// TwinCAT 3 PLC project iin_base
// Title: IIN_Base_T
// Company: IIN Solutions Oy
// Author: Author
// ProjectVersion: 0.0.3
// ProgramVersion: 3.1.4026.21
// libraries:
//   Tc2_Standard, * (Beckhoff Automation GmbH)
//   Tc2_System, * (Beckhoff Automation GmbH)
//   Tc2_Utilities, * (Beckhoff Automation GmbH)
//   VisuDialogs, * (System)
// project tree:
//   ALARMS/AlarmObserver/ I_AlarmObserver.TcIO
//   ALARMS/AppSupport/ FB_Interceptor.TcPOU, FB_StepperProgram.TcPOU, FC_GetLoggingId.TcPOU, FC_GetPositionWithId.TcPOU, FC_GetPosNrWithId.TcPOU, ST_INTERCEPTOR.TcDUT, ST_INTERCEPTOR_RESULT.TcDUT
//   ALARMS/DUT/ ST_ACTIVE_ALARM.TcDUT, ST_ALARM_BASE.TcDUT, ST_CLEAR_ALARM.TcDUT, ST_RAISE_ALARM.TcDUT
//   BASE/AdsUtils/ E_ADS_ERRORS.TcDUT, FC_GetAdsErrorCode.TcPOU, TL_ADS_ERRORS.TcTLO
//   BASE/ControlSignals/ FB_ControlSignalResets.TcPOU, FB_ControlSignalsV2.TcPOU, I_ControlSignals.TcIO, ST_CONTROL_SIGNALS_IN.TcDUT, ST_CONTROL_SIGNALS_OUT.TcDUT, ST_CONTROL_SIGNALS_SETTINGS.TcDUT, ST_CONTROL_SIGNALS_STATIC_SETTINGS.TcDUT, ST_CONTROL_SIGNALS_V2.TcDUT, TC_HMI_CS.TcDUT
//   BASE/CycleStartEnd/ FB_CycleEnd.TcPOU, FB_CycleStart.TcPOU, FC_GetCurrentCycleCount.TcPOU
//   BASE/FileUtils/ FC_FilePathGenerator.TcPOU
//   BASE/LocaleUtils/ E_REGIO_SELECTION.TcDUT, FB_GetLocalTimeAndDate.TcPOU, FB_TimeSync.TcPOU, FC_CallAtStart_EpochTime.TcPOU, FC_DateAndTimeToDt.TcPOU, FC_FormatTime.TcPOU, FC_GetEpochTime.TcPOU, FC_GetLocalDateAndTimeString.TcPOU, FC_GetLocalDateString.TcPOU, FC_GetLocalTimeString.TcPOU, FC_GetLocalTimeStringMinAccuracy.TcPOU, FC_GetLocalTimeStringSecAccuracy.TcPOU, FC_GetUsDateString.TcPOU, FC_NowAsDt.TcPOU, FC_TimeStringToDt.TcPOU
//   BASE/Misc/ COLORS.TcGVL, FB_Base.TcPOU, FB_BaseWithAlarmEvents.TcPOU, FB_BoolLogger.TcPOU, FB_BoolTrigger.TcPOU, FB_DelayedReset.TcPOU, FB_HandshakeDelay.TcPOU, FB_IntChangeTrigger.TcPOU, FB_IntLogger.TcPOU, FB_MemoryMonitor.TcPOU, FB_OneCycleSignalTof.TcPOU, FB_TofOnRtrig.TcPOU, FC_GetLocalAmsNetId.TcPOU, FC_GetLocalHostName.TcPOU, FC_GetMax3Arg.TcPOU, FC_GetMax3Lreals.TcPOU, FC_GetMax4Arg.TcPOU, FC_GetMin2Arg.TcPOU, FC_GetMin3Arg.TcPOU, FC_GetMin3Lreals.TcPOU, FC_GetMin4Arg.TcPOU, IING.TcGVL, ST_BASE_SETTINGS.TcDUT
//   BASE/NumberUtils/ AddREAL.TcPOU, DecINT.TcPOU, FC_CheckMinMaxInt.TcPOU, FC_CheckMinMaxReal.TcPOU, FC_KeepBetweenMinMax.TcPOU, FC_KeepBetweenMinMaxInt.TcPOU, FC_KeepRealBetweenMinMax.TcPOU, FC_LimitMaxReal.TcPOU, FC_LimitMinReal.TcPOU, FC_WithinMinMax.TcPOU, FC_WithinRange.TcPOU, IncINT.TcPOU, IncUDINT.TcPOU, IncUINT.TcPOU, IncULINT.TcPOU
//   BASE/Observer/ FB_GenericObserver.TcPOU, GVL_GENERIC_OBSERVER.TcGVL, ST_GENERIC_OBSERVER.TcDUT, ST_VALID_OBSERVERS.TcDUT
//   BASE/Persistency/ FB_Persistency.TcPOU, ST_PERSISTENCY_HMI.TcDUT, ST_PERSISTENCY_OUT.TcDUT, ST_PERSISTENCY_SERVICE.TcDUT, ST_PERSISTENCY_SETTINGS.TcDUT
//   BASE/PulsersBlinkers/ FB_Blink.TcPOU, FB_Blinkers.TcPOU, FB_Pulse.TcPOU, FB_Pulsers.TcPOU
//   BASE/StringUtils/ FC_2strConcatSeparator.TcPOU, FC_3strConcat.TcPOU, FC_3strConcatSeparator.TcPOU, FC_4strConcat.TcPOU, FC_4strConcatSeparator.TcPOU, FC_5strConcat.TcPOU, FC_5strConcatSeparator.TcPOU, FC_6strConcat.TcPOU, FC_6strConcatSeparator.TcPOU, FC_7strConcat.TcPOU, FC_7strConcatSeparator.TcPOU, FC_8strConcat.TcPOU, FC_8strConcatSeparator.TcPOU, FC_CharReplace.TcPOU, FC_FindLastOccurence.TcPOU, FC_InitializeNameAsNeeded.TcPOU, FC_IsBaseNameDefined.TcPOU, FC_LrealFormatter.TcPOU, FC_RealFormatter.TcPOU, FC_StringEmpty.TcPOU, FC_StringNotEmpty.TcPOU, FC_UintFormatter.TcPOU, IsStringEqualIgnoreCase.TcPOU
//   BASE/TypeDefinitions/ T_DEFAULT_STR.TcDUT, T_EVENT_CHAR_INDICATOR.TcDUT, T_HEART_BEAT.TcDUT, T_LONG_STR_512.TcDUT, T_SHORT_STR.TcDUT
//   DATA/DUT/ E_ALARM_REASON.TcDUT, E_ALARM_TYPE.TcDUT, E_DEVICE_TYPE.TcDUT, E_OPERATION_MODE.TcDUT, E_POS.TcDUT, E_PRIORITY.TcDUT, E_RESET_ORIGIN.TcDUT, T_DEVICE_ID.TcDUT
//   DATA/REPORTING/ DATA_REPORTER_BASE.TcGVL, FB_DummyDataReporter.TcPOU, FC_GetDataReporter.TcPOU, I_DataReporter.TcIO
//   LOGGING/ FC_GetLogger.TcPOU, LOGGER.TcGVL, NullLogger.TcPOU
//   LOGGING/FileLogger/ E_FILE_LOGGER_STEPS.TcDUT, E_FILE_SCANNER_STEPS.TcDUT, E_FILE_WRITER_STEPS.TcDUT, FB_FileLogger.TcPOU, FB_FileNameAndPath.TcPOU, FB_FileScannerV2.TcPOU, FB_FileWriterV2.TcPOU, ST_FILE_LOGGER_HMI.TcDUT, ST_FILE_LOGGER_SERVICE.TcDUT, ST_FILE_LOGGER_SETTINGS.TcDUT
//   LOGGING/GenericLogger/ FB_GenericLogger.TcPOU
//   LOGGING/NullLogger/ FB_NullLogger.TcPOU
//   LOGGING/Specs/ E_LOG_LEVEL.TcDUT, FB_LogLevel.TcPOU, I_Logger.TcIO, TL_LOG_LEVEL.TcTLO

// ---- ALARMS/AppSupport/ST_INTERCEPTOR.TcDUT
TYPE ST_INTERCEPTOR :
STRUCT
	check:	BOOL;
	desc:	T_SHORT_STR;
END_STRUCT
END_TYPE

// ---- ALARMS/AppSupport/ST_INTERCEPTOR_RESULT.TcDUT
TYPE ST_INTERCEPTOR_RESULT :
STRUCT
	clear:		BOOL;				// When TRUE, all is good 
	missing:	T_SHORT_STR;		// When clear is FALSE, this tells what is missing
END_STRUCT
END_TYPE

// ---- ALARMS/DUT/ST_ACTIVE_ALARM.TcDUT
TYPE ST_ACTIVE_ALARM EXTENDS ST_RAISE_ALARM:
STRUCT
	timestamp:				T_SHORT_STR;						// Timestamp when this occured
	epochTime:				ULINT;								// Needed for sorting purposes
	active:					BOOL;								// TRUE = currently active
END_STRUCT
END_TYPE

// ---- ALARMS/DUT/ST_ALARM_BASE.TcDUT
TYPE ST_ALARM_BASE :
STRUCT
	alarmType:			E_ALARM_TYPE := E_ALARM_TYPE.UNDEFINED;
	deviceType:			E_DEVICE_TYPE := E_DEVICE_TYPE.UNDEFINED;

	pos:				E_POS := E_POS.UNDEFINED;
	deviceId:			T_DEVICE_ID := IING.STRING_BLANK;
	
	// Unique ID generated when the alarm gets raised
	uniqueId:			ULINT;
	
	priority:			E_PRIORITY;
END_STRUCT
END_TYPE

// ---- ALARMS/DUT/ST_CLEAR_ALARM.TcDUT
TYPE ST_CLEAR_ALARM EXTENDS ST_ALARM_BASE :
STRUCT
END_STRUCT
END_TYPE

// ---- ALARMS/DUT/ST_RAISE_ALARM.TcDUT
TYPE ST_RAISE_ALARM EXTENDS ST_ALARM_BASE:
STRUCT
	givenDeviceName:		STRING;
	freeText:				STRING;
	subAlarmCode:			INT;
	
END_STRUCT
END_TYPE

// ---- BASE/AdsUtils/E_ADS_ERRORS.TcDUT
{attribute 'qualified_only'}
{attribute 'strict'}
TYPE E_ADS_ERRORS :
(
	// Global Error Codes
	NO_ERROR := 0,
	
	TARGET_PORT_NOT_FOUND := 6,
	
	TARGET_MACHINE_NOT_FOUND := 7,
	
	// General ADS Error Codes
	ADSERR_DEVICE_ERROR := 1792,
	
	ADSERR_DEVICE_SRVNOTSUPP := 1793,
	
	ADSERR_DEVICE_INVALIDGRP := 1794,
	
	ADSERR_DEVICE_INVALIDOFFSET := 1795,
	
	ADSERR_DEVICE_INVALIDACCESS := 1796,
	
	ADSERR_DEVICE_INVALIDSIZE := 1797,

	ADSERR_DEVICE_INVALIDDATA := 1798,

	ADSERR_DEVICE_NOTREADY := 1799,

	ADSERR_DEVICE_BUSY := 1800,

	ADSERR_DEVICE_INVALIDCONTEXT := 1801,

	ADSERR_DEVICE_NOMEMORY := 1802,
	
	ADSERR_DEVICE_INVALIDPARM := 1803,
	
	ADSERR_DEVICE_NOTFOUND := 1804,
	
	ADSERR_DEVICE_SYNTAX := 1805,
	
	ADSERR_DEVICE_INCOMPATIBLE := 1806,
	
	ADSERR_DEVICE_EXISTS := 1807,
	
	ADSERR_DEVICE_SYMBOLNOTFOUND := 1808,
	
	ADSERR_DEVICE_SYMBOLVERSIONINVAL := 1809,
	
	ADSERR_DEVICE_INVALIDSTATE := 1810,

	ADSERR_DEVICE_TRANSMODENOTSUPP := 1811,
	
	ADSERR_DEVICE_NOTIFYHNDINVALID := 1812,
	
	ADSERR_DEVICE_CLIENTUNKNOWN := 1813,
	
	ADSERR_DEVICE_NOMOREHDLS := 1814,
	
	ADSERR_DEVICE_INVALIDWATCHSIZE := 1815,
	
	ADSERR_DEVICE_NOTINIT := 1816,
	
	ADSERR_DEVICE_TIMEOUT := 1817,
	
	ADSERR_DEVICE_NOINTERFACE := 1818,
	
	ADSERR_DEVICE_INVALIDINTERFACE := 1819,
	
	ADSERR_DEVICE_INVALIDCLSID := 1820,
	
	ADSERR_DEVICE_INVALIDOBJID := 1821,
	
	ADSERR_DEVICE_PENDING := 1822,
	
	ADSERR_DEVICE_ABORTED := 1823,
	
	ADSERR_DEVICE_WARNING := 1824,
	
	ADSERR_DEVICE_INVALIDARRAYIDX := 1825,
	
	ADSERR_DEVICE_SYMBOLNOTACTIVE := 1826,
	
	ADSERR_DEVICE_ACCESSDENIED := 1827,
	
	ADSERR_DEVICE_LICENSENOTFOUND := 1828,
	
	ADSERR_DEVICE_LICENSEEXPIRED := 1829,
	
	ADSERR_DEVICE_LICENSEEXCEEDED := 1830,
	
	ADSERR_DEVICE_LICENSEINVALID := 1831,
	
	ADSERR_DEVICE_LICENSESYSTEMID := 1832,
	
	ADSERR_DEVICE_LICENSENOTIMELIMIT := 1833,
	
	ADSERR_DEVICE_LICENSEFUTUREISSUE := 1834,
	
	ADSERR_DEVICE_LICENSETIMETOLONG := 1835,
	
	ADSERR_DEVICE_EXCEPTION := 1836,
	
	ADSERR_DEVICE_LICENSEDUPLICATED := 1837,
	
	ADSERR_DEVICE_SIGNATUREINVALID := 1838,
	
	ADSERR_DEVICE_CERTIFICATEINVALID := 1839,
	
	ADSERR_CLIENT_ERROR := 1856,
	
	ADSERR_CLIENT_INVALIDPARM := 1857,
	
	ADSERR_CLIENT_LISTEMPTY := 1858,
	
	ADSERR_CLIENT_VARUSED := 1859,
	
	ADSERR_CLIENT_DUPLINVOKEID := 1860,
	
	ADSERR_CLIENT_SYNCTIMEOUT := 1861,
	
	ADSERR_CLIENT_W32ERROR := 1862,
	
	ADSERR_CLIENT_TIMEOUTINVALID := 1863,
	
	ADSERR_CLIENT_PORTNOTOPEN := 1864,
	
	ADSERR_CLIENT_NOAMSADDR := 1872,
	
	ADSERR_CLIENT_SYNCINTERNAL := 1873,
	
	ADSERR_CLIENT_ADDHASH := 1874,
	
	ADSERR_CLIENT_REMOVEHASH := 1875,
	
	ADSERR_CLIENT_NOMORESYM := 1876,
	
	ADSERR_CLIENT_SYNCRESINVALID := 1877,

	TODO := 9999
	
);
END_TYPE

// ---- BASE/ControlSignals/ST_CONTROL_SIGNALS_IN.TcDUT
TYPE ST_CONTROL_SIGNALS_IN :	// The raw control signals (auto/manual/service/...), do not use in your application
STRUCT
	manualMode:			BOOL;	// Auto/Manual
	serviceMode:		BOOL;
	pauseRequest:		BOOL;	// Will let ongoing operations finish nicely, When TRUE = must go to Pause, when FALSE, may continue
	stopImmediately:	BOOL;	// Placeholder for later use
	restart:			BOOL;	// Placeholder for later use
	
	reset:				BOOL;	// Reset button (a single PLC pulse will be generated from this)
	hardReset:			BOOL;	// Hard reset button (a single PLC pulse will be generated from this)

//	safetyAreaOk:		BOOL;	// Estop and doors are 'safe' = possible to drive in AUTO
	
	externalReset:		BOOL;	// External reset coming from FB_ControlSignalsV2/iExternalReset
	autoReset:			BOOL;	// Auto reset coming from FB_ControlSignalsV2/iAutoReset
END_STRUCT
END_TYPE

// ---- BASE/ControlSignals/ST_CONTROL_SIGNALS_OUT.TcDUT
TYPE ST_CONTROL_SIGNALS_OUT :	// Control signals (auto/manual/service/...) for use in programs 
STRUCT
	auto:						BOOL;	// TRUE when in automatic mode
	manual:						BOOL;	// TRUE when in manual mode
	service:					BOOL;	// TRUE when in service mode
	
	autoPulse:					BOOL;	// Single PLC cycle pulse when switching to AUTO
	manualPulse:				BOOL;	// Single PLC cycle pulse when switching to MANUAL
	servicePulse:				BOOL;	// Single PLC cycle pulse when switching to SERVICE
	
	autoOffPulse:				BOOL;	// TRUE for 1 PLC cycle when switching AUTO OFF
	manualOffPulse:				BOOL;	// TRUE for 1 PLC cycle when switching MANUAL OFF
	serviceOffPulse:			BOOL;	// TRUE for 1 PLC cycle when switching SERVICE OFF
	
	pauseRequest:				BOOL;	// TRUE when pause requested
	stopImmediately:			BOOL;	// Single PLC cycle pulse
	restart:					BOOL;	// Single PLC cycle pulse

	resetPulse:					BOOL;	// Single PLC cycle pulse for resetting (after error)
	hardResetPulse:				BOOL;	// Single PLC cycle pulse for hard reset (wipe out everything)
	
	extendedResetPulse:			BOOL;	// Extended reset pulse, eg. for external systems
	extendedHardResetPulse:		BOOL;	// Extended hard reset pulse, eg. for external systems
	
	externalManualActive:		bool;
	failingToSwitchToAuto:		BOOL;
END_STRUCT
END_TYPE

// ---- BASE/ControlSignals/ST_CONTROL_SIGNALS_SETTINGS.TcDUT
TYPE ST_CONTROL_SIGNALS_SETTINGS EXTENDS ST_BASE_SETTINGS:
STRUCT
	// All of them are under VAR_STAT
END_STRUCT
END_TYPE

// ---- BASE/ControlSignals/ST_CONTROL_SIGNALS_STATIC_SETTINGS.TcDUT
TYPE ST_CONTROL_SIGNALS_STATIC_SETTINGS:
STRUCT
	resetTime:						TIME := IING.RESET_TIME;
	hardResetTime:					TIME := IING.HARD_RESET_TIME;
	serviceResetTime:				TIME := IING.AUTO_SERVICE_RESET_TIME;	// Time after which service mode is swithced OFF
	extendedResetPulseDuration:		TIME := IING.EXTENDED_RESET_PULSE_DURATION;
END_STRUCT
END_TYPE

// ---- BASE/ControlSignals/ST_CONTROL_SIGNALS_V2.TcDUT
TYPE ST_CONTROL_SIGNALS_V2 :	// Control signals (auto/manual/service/...) for use in programs 
STRUCT
	in:				 	ST_CONTROL_SIGNALS_IN;
	out:				ST_CONTROL_SIGNALS_OUT;
	
	settings:			REFERENCE TO ST_CONTROL_SIGNALS_SETTINGS;
	staticSettings:		REFERENCE TO ST_CONTROL_SIGNALS_STATIC_SETTINGS;
END_STRUCT
END_TYPE

// ---- BASE/ControlSignals/TC_HMI_CS.TcDUT
TYPE TC_HMI_CS :
STRUCT
	out:		ST_CONTROL_SIGNALS_OUT;
	in:	ST_CONTROL_SIGNALS_IN;
END_STRUCT
END_TYPE

// ---- BASE/LocaleUtils/E_REGIO_SELECTION.TcDUT
{attribute 'qualified_only'}
{attribute 'strict'}
TYPE E_REGIO_SELECTION :
(
	USA := 0,
	EUROPE
);
END_TYPE

// ---- BASE/Misc/ST_BASE_SETTINGS.TcDUT
TYPE ST_BASE_SETTINGS :
STRUCT
	name:			T_SHORT_STR := IING.STRING_BASE_SETTINGS_INITIAL_NAME;
	doHide:			BOOL := TRUE;
END_STRUCT
END_TYPE

// ---- BASE/Observer/ST_GENERIC_OBSERVER.TcDUT
TYPE ST_GENERIC_OBSERVER :
STRUCT
	who:		T_SHORT_STR;			// Unique identifier of this observer
	observer:	POINTER TO BYTE;		// Interface CASTed to a generic POINTER, to be CASTed back in your application
END_STRUCT
END_TYPE

// ---- BASE/Observer/ST_VALID_OBSERVERS.TcDUT
TYPE ST_VALID_OBSERVERS :
STRUCT
	cnt:		INT;
	observers:	ARRAY[0..GVL_GENERIC_OBSERVER.OBSERVER_CNT-1] OF ST_GENERIC_OBSERVER;
END_STRUCT
END_TYPE

// ---- BASE/Persistency/ST_PERSISTENCY_HMI.TcDUT
TYPE ST_PERSISTENCY_HMI :
STRUCT
	service:		REFERENCE TO ST_PERSISTENCY_SERVICE;
	settings:		REFERENCE TO ST_PERSISTENCY_SETTINGS;
	out:			REFERENCE TO ST_PERSISTENCY_OUT;
END_STRUCT
END_TYPE

// ---- BASE/Persistency/ST_PERSISTENCY_OUT.TcDUT
TYPE ST_PERSISTENCY_OUT :
STRUCT
	busy:					BOOL;
	error:					BOOL;
	beckhoffErrorId:		UDINT;
	errorIdEnum:			E_ADS_ERRORS;
END_STRUCT
END_TYPE

// ---- BASE/Persistency/ST_PERSISTENCY_SERVICE.TcDUT
TYPE ST_PERSISTENCY_SERVICE :
STRUCT
	saveNow:		BOOL;
END_STRUCT
END_TYPE

// ---- BASE/Persistency/ST_PERSISTENCY_SETTINGS.TcDUT
TYPE ST_PERSISTENCY_SETTINGS :
STRUCT
	port:				UINT := 851;	
	autoSave:			BOOL := TRUE;
	saveInterval:		TIME := T#12H;
END_STRUCT
END_TYPE

// ---- BASE/TypeDefinitions/T_DEFAULT_STR.TcDUT
TYPE T_DEFAULT_STR : STRING(255); END_TYPE		// Use this instead of STRING which is 80 chars only

// ---- BASE/TypeDefinitions/T_EVENT_CHAR_INDICATOR.TcDUT
TYPE T_EVENT_CHAR_INDICATOR : STRING(1); END_TYPE

// ---- BASE/TypeDefinitions/T_HEART_BEAT.TcDUT
TYPE T_HEART_BEAT : UDINT; END_TYPE		// Signal used to check the heart beat (over ADS)

// ---- BASE/TypeDefinitions/T_LONG_STR_512.TcDUT
TYPE T_LONG_STR_512 : STRING(512); END_TYPE		// Use this instead of STRING which is 80 chars only

// ---- BASE/TypeDefinitions/T_SHORT_STR.TcDUT
TYPE T_SHORT_STR : STRING(80); END_TYPE		// Use this for 'shorter' string

// ---- DATA/DUT/E_ALARM_REASON.TcDUT
{attribute 'qualified_only'}

{attribute 'to_string'}
TYPE E_ALARM_REASON :
(
	UNDEFINED,
	
	NO_COOLING,
	
	OVERLOAD,
	
	WRONG_ITEM,
	
	WRONG_DIMENSION,
	
	WRONG_ORIENTATION,
	
	STUCK,
	
	NO_PRESSURE,
	
	OTHER,	
	
	MUST_BE_LAST	// ALWAYS KEEP THIS LAST!!!
	
);
END_TYPE

// ---- DATA/DUT/E_ALARM_TYPE.TcDUT
{attribute 'qualified_only'}
{attribute 'to_string'}
TYPE E_ALARM_TYPE :
(
	UNDEFINED := 0,

	// An operation took too long to complete
	TIME_OUT,

	// A sensor is blocked
	SENSOR_BLOCKED,
	
	// Bad request, eg. asking to open and close a cylinder at the same time 
	BAD_REQUEST,
	
	// Overload from eg. a fuse or servo drive
	OVERLOAD,
	
	// A component is overheating
	OVERHEAT,

	// Collision detected
	COLLISION,
	
	// Regular servo error
	SERVO_ERROR,
	
	// Positioning error
	POSITIONING_ERROR,
	
	// Velocity error
	VELOCITY_ERROR,
	
	MOVE_RELATIVE_ERROR,
	
	// Jogging error
	JOGGING_ERROR,

	// Probing error	
	PROBING_ERROR,
	
	// Gearing error
	GEARING_ERROR,
	
	GEAR_IN_ERROR,
	
	GEAR_OUT_ERROR,
	
	// Measurement of a member/truss did not match the WP length
	DIMENSION_MISMATCH,
	
	// Buffer station or robots get values not in the allowed work area
	WRONG_COORDINATES,
	
	// Member id (or eventId) mismatch, plate mismatch
	ITEM_MISMATCH,
	
	ESTOP,
	
	BELOW_MIN,
	
	ABOVE_MAX,
	
	// Communication error
	COMM_ERROR,
	
	MISSING_PART,
	
	HOMING_ERROR,
	
	ZEROING_ERROR,
	
	TOOL_DROP,
	
	SAFETY,
	
	DOCKING_STATION_ERROR,
	
	PARSE_ERROR,
	
	TOOL_CHANGER_ERROR,
	
	// Sequence expects something but this is not fullfilled
	WRONG_STATE,
	
	HOMING_NOT_ENABLED,
	
	// Eg, not supported settings (nor head, nor tail selection)
	CONFIGURATION_ERROR,

	FORCING,			// Used with the Forcing alarm manager
	
	NO_POWER,			// Power supply 'OFF'
	
	INTERRUPTION,		// Something got interrupted/stopped, eg. STOPMESS in robot

	TASK_DIED,			// Eg. submit interpreter not running
	
	SIMULATION_ACTIVE,
	
	STICKY_BUTTON,		// Eg. a button is sticky (PLC HMI)
	
	SAFE_TORQUE_OFF,	// STO active, eg, freq drive or servo
	
	FREQ_DRIVE_ERROR,	// Any kind of frequence related error

	START_CONDITIONS_NOT_MET,
	
	MISC,
	
	OUT_OF_RANGE,
	
	CLOGGED,					// Eg. filter clogged
	
	MISSING,					// Eg. air pressure missing
	
	OPEN,						// Eg. a door is open
	
	PREMATURE_DETECTION,		// Probing ready before slowing down conveyor
	
	TRIGGERED,					// Safety scanner got triggered
	
	LOW_VALUE,					// eg. speed setting rather low, intentional?
	
	DEVIATION_DETECTED,			// AI and AO settings not matching (enfield)
	
	OVERSHOOTING,				// Servo is overshooting (then reversing)
	
	SENSOR_BROKEN,				// AI readings not possible
	
	ROBOT_APP_ERROR,			// Robot sends us some error code (probably calculation/e1 related)
	
	VACUUM_MISSING,				// Vacuum is missing
	
	MANUAL_MODE,				// Device is in manual
	
	EDM,						// External Device Monitoring
	
	CLOSED,						// Eg. a (gantry) door is closed
	
	WAITING_CONFIRMATION,
	
	SUPER_POWERS,
	
	END //63
	
);
END_TYPE

// ---- DATA/DUT/E_DEVICE_TYPE.TcDUT
{attribute 'qualified_only'}

{attribute 'to_string'}
TYPE E_DEVICE_TYPE :
(
	UNDEFINED,
	
	// Special case for alarm handler	
	ACCEPT_ANY,
	
	MOTOR,					// Direct drive motor

	SERVO,					// Servo drive
	
	FREQ_DRIVE,				// 'TAMU'

	FUSE,
	
	RELAIS,
	
	VALVE,
	
	CYLINDER,
	
	HYDRAULIC,
	
	SCANNER,				// Eg. sick scanner		

	PRINTER,		
	
	DOOR,					// Eg. Safety door
	
	ESTOP,
	
	BRAKE,
	
	PSU,
	
	FILTER,					// Eg. oil/air filter
	
	CONVEYOR,
	
	COMM_CHANNEL,
	
	TURN_TABLE,
	
	MISC,
	
	ROBOT,
	
	MAGNET,
	
	SENSOR,		// Use this for
	
	SPEED_CONTROL,	// Device speed
	
	TOOL_CHANGER,
	
	BUTTON_BOX,
	
	PNEUMATIC,
	
	SAFETY,
	
	ENCODER,
	
	SEQUENCE,
	
	CONTROL_SIGNALS,
	
	END	// ALWAYS KEEP THIS LAST!!!
);
END_TYPE

// ---- DATA/DUT/E_OPERATION_MODE.TcDUT
{attribute 'qualified_only'}
{attribute 'strict'}
{attribute 'to_string'}
TYPE E_OPERATION_MODE :
(
	UNDEFINED,
	
	AUTO,

	MANUAL,
	
	MUST_BE_LAST	// ALWAYS KEEP THIS LAST!!!
);
END_TYPE

// ---- DATA/DUT/E_POS.TcDUT
{attribute 'qualified_only'}
{attribute 'to_string'}
TYPE E_POS :			// Position numbers
(
	UNDEFINED := 0,
	
	// Special case for alarm handler	
	ACCEPT_ANY := 1,

	MAIN :=		10,
	

	
	
	MUST_BE_LAST	// ALWAYS KEEP THIS LAST!!!
);
END_TYPE

// ---- DATA/DUT/E_PRIORITY.TcDUT
{attribute 'qualified_only'}
{attribute 'strict'}
{attribute 'to_string'}
TYPE E_PRIORITY :
(
	UNDEFINED,
	
	LOW,
	
	MEDIUM,
	
	HIGH,
	
	MUST_BE_LAST	// ALWAYS KEEP THIS LAST!!!
);
END_TYPE

// ---- DATA/DUT/E_RESET_ORIGIN.TcDUT
{attribute 'qualified_only'}
{attribute 'strict'}
{attribute 'to_string'}
TYPE E_RESET_ORIGIN :
(
	UNDEFINED := 0,
	
	CONTROL_AREA_MANUAL,	// Operator presses reset on the control signal
	
	CONTROL_AREA_AUTO,		// Automatic (external) reset, eg. doors were closed and a reset was triggered

	EXTERNAL,				// Through FB input, eg. hard wired button or banner reset
	
	ALARM_SPECIFIC			// Specific device/alarm reset 
);
END_TYPE

// ---- DATA/DUT/T_DEVICE_ID.TcDUT
TYPE T_DEVICE_ID : STRING; END_TYPE

// ---- LOGGING/FileLogger/E_FILE_LOGGER_STEPS.TcDUT
{attribute 'qualified_only'}
{attribute 'strict'}
TYPE E_FILE_LOGGER_STEPS :
(
	WAIT_ACTIVITY := 0,
	
	CHECK_SIZE,
	
	CLOSE_FILE,
	
	SCAN_FOLDER,
	
	ITERATE_FILES,
	
	RENAME_FILE,
	
	RENAME_FILE_ERROR,
	
	END
);
END_TYPE

// ---- LOGGING/FileLogger/E_FILE_SCANNER_STEPS.TcDUT
{attribute 'qualified_only'}
{attribute 'strict'}
TYPE E_FILE_SCANNER_STEPS :
(
	IDLE := 0,
	
	SCAN,
	
	STORE_FILE,
	
	DONE,
	
	ERROR,
	
	END
);
END_TYPE

// ---- LOGGING/FileLogger/E_FILE_WRITER_STEPS.TcDUT
{attribute 'qualified_only'}
{attribute 'strict'}
TYPE E_FILE_WRITER_STEPS :
(
	IDLE := 0,
	
	OPEN_FILE,
	
	WAIT_DATA,
	
	WRITE_LINE,

	CHECK_FILE,
	
	CLOSE_FILE,
	
	CLEANUP,
	
	OPENING_ERROR,
	
	TELL_ERROR,
	
	WRITING_ERROR,
	
	CLOSING_ERROR,
	
	END
);
END_TYPE

// ---- LOGGING/FileLogger/ST_FILE_LOGGER_HMI.TcDUT
TYPE ST_FILE_LOGGER_HMI :
STRUCT
	// Modifiable from HMI
	service:					REFERENCE TO ST_FILE_LOGGER_SERVICE;
	settings:					REFERENCE TO ST_FILE_LOGGER_SETTINGS;	
	controlSignals:				REFERENCE TO ST_CONTROL_SIGNALS_IN;

	amsNetId:					T_AmsNetId;
	fileNameAndPath:			T_DEFAULT_STR;					// VISU helper
	tracingOn:					BOOL;							// TRUE when log level is trace
	tracingTimeExpired:			TIME;							// Amount of trace time expired
	autoResetOn:				BOOL;							// TRUE when auto reset is ON
	outResetTimer:				TIME;							// After this time, auto reset will be done
	error:						BOOL;							// TRUE if a file writing error occurs
	adsErrorCode:				E_ADS_ERRORS;
	fileWriterRecordCnt:		UDINT;
	fileWriterBytesUsed:		UDINT;
	fileWriterOverflowCount:	UDINT;							// How many times we were not able to write all data to the file (due to internal memory constraints)
END_STRUCT
END_TYPE

// ---- LOGGING/FileLogger/ST_FILE_LOGGER_SERVICE.TcDUT
TYPE ST_FILE_LOGGER_SERVICE :
STRUCT
	doFileFlush:			BOOL;							// Set TRUE when flush is wanted
END_STRUCT
END_TYPE

// ---- LOGGING/FileLogger/ST_FILE_LOGGER_SETTINGS.TcDUT
TYPE ST_FILE_LOGGER_SETTINGS EXTENDS ST_BASE_SETTINGS:
STRUCT
	logLevel:				E_LOG_LEVEL := E_LOG_LEVEL.ERROR;	// The current log level
	maxFileSizeMB:			DINT := 10;							// File size (MB) after which, the log file will be rolled over
	enableMaxTracingTime:	BOOL := FALSE;						// When TRUE, TRACING can be switched off automatically
	maxTracingTime:			TIME := T#1H;						// Max amount of time TRACING will be active, after this DEBUG becomes activeEND_STRUCT
	enableAutoReset:		BOOL := TRUE;						// When TRUE, write errors will be reset automatically
	autoResetTime:			TIME := T#1H;						// After this amount of time, an error reset will be done
END_STRUCT
END_TYPE

// ---- LOGGING/Specs/E_LOG_LEVEL.TcDUT
{attribute 'qualified_only'}
{attribute 'strict'}
{attribute 'to_string'}
TYPE E_LOG_LEVEL :
(
	TRACE := 0,			// Use for hard to find problems = tracing problems, this will generate a log of data
	
	DEBUG,			// Debug logging (steps)
	
	INFO,			// Use for informational messages
	
	WARN,			// Use for warnings
	
	ERROR,			// Use for errors/alarms

	OFF			// Nothing will be logged
);
END_TYPE

// ---- BASE/Misc/COLORS.TcGVL
{attribute 'qualified_only'}
{attribute 'global_init_slot' := '40001'}
VAR_GLOBAL CONSTANT
	LILA:	DWORD := 16#FF0F0DF1;
	PINK:	DWORD := 16#FFE943D4;
	ORANGE:	DWORD := 16#FFFFCC00;
	BLUE :	DWORD := 16#FF0000FF;
	RED	:	DWORD := 16#FFFF0000;
	YELLOW:	DWORD := 16#FFFFFF00;
	GREEN:	DWORD := 16#FF00FF00;
	GREY:	DWORD := 16#FFC0C0C0;
	WHITE:	DWORD := 16#FFFFFFFF;
	BLACK:	DWORD := 16#FF000000;	
END_VAR

// ---- BASE/Misc/IING.TcGVL
{attribute 'qualified_only'}
{attribute 'global_init_slot' := '40002'}
VAR_GLOBAL
	epochtime :						ULINT;				// Epoch time (milliseconds)
	localSystemTime:				TIMESTRUCT;			// Local system time
	localDateString:				T_SHORT_STR;		// Local date string, eg. '27:5:2019'. Use E_REGIO_SELECTION at FB_CycleStart for a different format.
	usDateString:					T_SHORT_STR;		// US style date string, especially usefull for naming log files
	localTimeString:				T_SHORT_STR;		// Local time as string, eg. '15:58:40:302'
	localDateAndTimeString:			T_SHORT_STR;		// Local date and time as string,  eg. '27:5:2019 15:58:40:302'. Use E_REGIO_SELECTION at FB_CycleStart for a different format.
	localHostName:					T_DEFAULT_STR;		// Local hostname
	localAmsNetId:					T_AmsNetId;			// Local AMS net id
	localTimeSecAccuracy:			T_SHORT_STR;		// Local time as string, eg. '15:58:40', seconds accuracy
	localTimeMinAccuracy:			T_SHORT_STR;		// Local time as string, eg. '15:58', minutes accuracy
	iso8601Time:					T_SHORT_STR;		// Time in ISO 8601 format
	
	cycleTime:						ULINT;				// Current PLC cycle time in msec
	cycleStart:						BOOL;				// TRUE during first PLC cycle
	lastPlcRestart:					T_SHORT_STR;		// Timestamp of last PLC restart
	dayHasChanged:					BOOL;				// TRUE for 1 PLC cycle when a day change occurs

	// Blinkers, usefull for making a light beacon blink
	blink100Ms:						BOOL;			// 100ms blinker  
	blink500Ms:						BOOL;			// 500ms blinker
	blink1S:						BOOL;			// 1S blinker
	blink2S:						BOOL;			// 2S blinker
	blink5S:						BOOL;			// 5S blinker
	blink10S:						BOOL;			// 10S blinker
	
	invertedBlink100Ms:				BOOL;			// Inverted 100ms blinker
	invertedBlink500Ms:				BOOL;			// Inverted 500ms blinker
	invertedBlink1S:				BOOL;			// Inverted 1S blinker
	invertedBlink2S:				BOOL;			// Inverted 2S blinker
	invertedBlink5S:				BOOL;			// Inverted 5S blinker
	invertedBlink10S:				BOOL;			// Inverted 10S blinker
 
	// 1 'PLC cycle' long pulsers 
	pulse100Ms:						BOOL;
	pulse500Ms:						BOOL;
	pulse1S:						BOOL;
	pulse2S:						BOOL;
	pulse10S:						BOOL;
	pulse30S:						BOOL;
	pulse1M:						BOOL;
	pulse1H:						BOOL;
	
	STRING_EMPTY_NON_CONSTANT:		T_SHORT_STR := '';			// Some VISUs want write access
	cycleCounter:					UDINT;			// Gets incremented each PLC cycle
	adsPort:						UINT;			// The ADS port we are running on
	
	simulatorActive:				BOOL;		// TRUE when running in simulation mode (TC project variant 'simulator')
	pointerSize:					UINT;		// Number of bytes for a pointer (=size)
END_VAR

VAR_GLOBAL CONSTANT
	TIME_OFFSET_1601 : 				ULINT := 11644472389000;	// Jan 01, 1601 (gotten from online millisecond calculator)
	TIME_OFFSET_20MINS :			ULINT := 20 *60 *1000;		// 1601 offset is 20 mins WRONG!
	EPOCH_CORRECTION :				ULINT := TIME_OFFSET_1601 + TIME_OFFSET_20MINS;		// Correction to get proper EPOCH timestamp instead of Beckhoff timestamp
	
	STRING_BLANK:					T_SHORT_STR := '';				// Use this instead of '', renamed from EMPTY->BLANK since same string exist in Beckhoff libs
	STRING_COLON: 					T_SHORT_STR := ':';				// Use this instead of ':'
	STRING_SPACE: 					T_SHORT_STR := ' ';				// Use this instead of ' '
	STRING_UNDERSCORE:				T_SHORT_STR := '_';				// Use this instead of '_'
	STRING_DASH:					T_SHORT_STR := '-';				// Use this instead of '-'
	STRING_COMMA:					T_SHORT_STR := ',';				// Use this instead of ','
	STRING_STAR:					T_SHORT_STR := '*';				// Use this instead of '*'
	STRING_SLASH:					T_SHORT_STR := '/';				// Use this instead of '/'
	STRING_BACKSLASH:				T_SHORT_STR := '\';				// Use this instead of '\'
	STRING_SQUARE_BRACKET_OPEN:		T_SHORT_STR := '[';				// Use this instead of '['
	STRING_SQUARE_BRACKET_CLOSE:	T_SHORT_STR := ']';				// Use this instead of ']'
	STRING_DOT:						T_SHORT_STR := '.';				// Use this instead of '.'
	STRING_PIPE:					T_SHORT_STR := '|';				// Use this instead of '|'
	STRING_AM:						T_SHORT_STR := 'AM';			// Use for time formatting
	STRING_PM:						T_SHORT_STR := 'PM';			// Use for time formatting
	STRING_BASE_SETTINGS_INITIAL_NAME:	T_SHORT_STR := '???';	// Initial name for the base setting
	STRING_EQUALS:					T_SHORT_STR := '=';				// Use this instead of '='
	STRING_EXCLAMATION:				T_SHORT_STR := '!';				// Use this instead of '!'
	STRING_UNDEFINED:				STRING := 'undefined';
	
	
	
	STRING_LINE_FEED:				T_SHORT_STR := '$0A';			// Use this when adding a line feed (eg. file handling)
	
	STRING_80_CHARS:				T_SHORT_STR := '0123456789012345678901234567890123456789012345678901234567890123456789012345678_';	// Use this for testing string functions (string by default is 80 chars only)
	STRING_TODO:					T_SHORT_STR := 'TODO';
	
	ADS_WRITE_TIMEOUT:				TIME := T#1S;				// Default ADS time-out for our applications
	ADS_WRITE_RETRIES:				UDINT := 3;					// Default number of ADS retries
	ADS_DEFAULT_PORT:				T_AmsPort := 851;			// Default ADS port (for 1st PLC)
	ADS_MB_INDEX_GROUP:				UDINT := 16#4020;			// ADS MB index group
	
	IDX_UNDEFINED:					INT := -1;					// Use this to make an array index invalid (instead of just 0)
	INVALID_UINT:					INT := -1;					// Use this to make an UINT invalid (instead of just 0)
	
	RESET_TIME:						TIME := T#100MS;			// Normal reset default time/delay
	HARD_RESET_TIME:				TIME := T#1S;				// Hard reset default time/delay
	AUTO_SERVICE_RESET_TIME:		TIME := T#5M;				// Time after which service mode is switched OFF
	EXTENDED_RESET_PULSE_DURATION:	TIME := T#250MS;
	SERVO_POWER_SAVINGS_TIME:		TIME := T#5M;				// Automatic powering down of a SERVO	
	
	BITS_IN_WORD:					UINT := 16;					// Number of bits in a WORD
	BITS_IN_DWORD:					UINT := 32;					// Number of bits in a DWORD
	
	FULL_SPEED:						REAL := 100.0;				// Use this as the default velocity override speed
	
	ZERO_POINTER:					UDINT := 0;					// Use this to 'null' a pointer/reference
	ONE_INCH:						LREAL := 25.4;				// One inch

	ONE_KBYTE:						DINT := 1024;				// One kilobyte in bytes	
	ONE_MBYTE:						DINT := 1048576;			// One megabyte in bytes
	
	MAX_UDINT:						UDINT := 16#FFFFFFFF;		// Biggest possible UDINT
	MAX_INT:						INT := 32767;				// Max value for an INT

	EVENT_INDICATION_NONE:			T_EVENT_CHAR_INDICATOR := STRING_BLANK;
	EVENT_INDICATION_WARNING:		T_EVENT_CHAR_INDICATOR := 'W';
	EVENT_INDICATION_ALARM:			T_EVENT_CHAR_INDICATOR := 'A';	
END_VAR

// ---- BASE/Observer/GVL_GENERIC_OBSERVER.TcGVL
{attribute 'qualified_only'}
VAR_GLOBAL CONSTANT
	OBSERVER_CNT:	INT := 5;
END_VAR

// ---- DATA/REPORTING/DATA_REPORTER_BASE.TcGVL
{attribute 'qualified_only'}
VAR_GLOBAL
	dummyReporter:		FB_DummyDataReporter;
	defaultReporter:	I_DataReporter;
END_VAR

// ---- LOGGING/LOGGER.TcGVL
{attribute 'qualified_only'}
VAR_GLOBAL
	nullLogger:				FB_NullLogger;					// DEV 0 logger
	defaultLogger:			I_Logger;	
END_VAR

// ---- ALARMS/AlarmObserver/I_AlarmObserver.TcIO
INTERFACE I_AlarmObserver

METHOD PUBLIC cleared : BOOL		// Called when an alarm is cleared
VAR_INPUT
	iAlarm:	ST_CLEAR_ALARM;
END_VAR
END_METHOD

METHOD PUBLIC raised : BOOL		// Called when an alarm is raised
VAR_INPUT
	iAlarm:	ST_ACTIVE_ALARM;
END_VAR
END_METHOD

END_INTERFACE

// ---- BASE/ControlSignals/I_ControlSignals.TcIO
INTERFACE I_ControlSignals

METHOD ic_getControlSignalsOutPtr : POINTER TO ST_CONTROL_SIGNALS_OUT
END_METHOD

METHOD PUBLIC ic_getControlSignalsPtr : POINTER TO ST_CONTROL_SIGNALS_V2
END_METHOD

METHOD PUBLIC ic_isInAuto : BOOL
END_METHOD

METHOD PUBLIC ic_isInPause : BOOL
END_METHOD

METHOD PUBLIC ic_switchToAuto
END_METHOD

METHOD ic_unPause
END_METHOD

END_INTERFACE

// ---- DATA/REPORTING/I_DataReporter.TcIO
INTERFACE I_DataReporter		// Interface for all data/mqtt reporting calls.
	// Idea is to keep logic away from the project/application, also reporting can be done in several ways, such as mqtt

METHOD PUBLIC ic_deviceSpeedChanged	// To be called when the (device) speed changes
VAR_INPUT
	iPos:			E_POS;				// Position enumerate
	iMiscArea:		T_SHORT_STR;		// Safety or misc area enumerate (string). If defined/non-empty, use this instead of iPos
	iNew:			INT;				// The new speed value
END_VAR
END_METHOD

METHOD PUBLIC ic_initializeDone	// To be called when a initialization (aka hard reset) is done
VAR_INPUT
	iPos:			E_POS;				// The position
	iMiscArea:		T_SHORT_STR;		// Safety or misc area enumerate (string). If defined/non-empty, use this instead of iPos
	iOrigin:		E_RESET_ORIGIN;	
END_VAR
END_METHOD

METHOD PUBLIC ic_operationModeChanged	// To be called when the control signal operation mode changes
VAR_INPUT
	iPos:			E_POS;				// The position
	iMiscArea:		T_SHORT_STR;		// Safety or misc area enumerate (string). If defined/non-empty, use this instead of iPos
	iNew:			E_OPERATION_MODE;	// New operation mode
END_VAR
END_METHOD

METHOD PUBLIC ic_resetDone	// To be called when the control signal operation mode changes
VAR_INPUT
	iPos:			E_POS;				// The position
	iMiscArea:		T_SHORT_STR;		// Safety or misc area enumerate (string). If defined/non-empty, use this instead of iPos
	iOrigin:		E_RESET_ORIGIN;
	iResetKeyLabel:	T_SHORT_STR;		// What reset key was pressed
END_VAR
END_METHOD

METHOD PUBLIC ic_serviceStateChanged		// To be called when the (control signal) service state changes
VAR_INPUT
	iPos:			E_POS;				// The position
	iMiscArea:		T_SHORT_STR;		// Safety or misc area enumerate (string). If defined/non-empty, use this instead of iPos
	iState:			BOOL;				// TRUE = service activated, FALSE = service deactivated
END_VAR
END_METHOD

END_INTERFACE

// ---- LOGGING/Specs/I_Logger.TcIO
INTERFACE I_Logger		// Generic interface for logging 'data', logging can be done to file/HMI/MQTT and depends on the implementation

METHOD PUBLIC debug : BOOL	// Logs the data with log level 'DEBUG'
VAR_INPUT
	iData:		T_DEFAULT_STR;						// Data to be logged, limited to 255 characters
END_VAR
END_METHOD

METHOD PUBLIC deregister : BOOL
VAR_INPUT
	iWho:				T_SHORT_STR;
END_VAR
END_METHOD

METHOD PUBLIC doLog : BOOL	// Logs the data with log level iLevel
VAR_INPUT
	iData:		T_DEFAULT_STR;						// Data to be logged, limited to 255 characters
	iLevel:		E_LOG_LEVEL := E_LOG_LEVEL.ERROR;	// Log level
END_VAR
END_METHOD

METHOD PUBLIC error : BOOL	// Logs the data with log level 'ERROR'
VAR_INPUT
	iData:		T_DEFAULT_STR;						// Data to be logged, limited to 255 characters
END_VAR
END_METHOD

METHOD PUBLIC info : BOOL	// Logs the data with log level 'INFO'
VAR_INPUT
	iData:		T_DEFAULT_STR;						// Data to be logged, limited to 255 characters
END_VAR
END_METHOD

METHOD PUBLIC register : BOOL
VAR_INPUT
	iWho:		T_SHORT_STR;
	iObserver:	I_Logger;
END_VAR
END_METHOD

METHOD PUBLIC trace : BOOL	// Logs the data with log level 'TRACE'
VAR_INPUT
	iData:		T_DEFAULT_STR;						// Data to be logged, limited to 255 characters
END_VAR
END_METHOD

METHOD PUBLIC warn : BOOL	// Logs the data with log level 'WARN'
VAR_INPUT
	iData:		T_DEFAULT_STR;						// Data to be logged, limited to 255 characters
END_VAR
END_METHOD

END_INTERFACE

// ---- BASE/CycleStartEnd/FB_CycleStart.TcPOU
FUNCTION_BLOCK FB_CycleStart		// Must always be the 1st call in PLC MAIN, ensures other functions/globals are available 
VAR_INPUT
	iRegioSelection:		E_REGIO_SELECTION := E_REGIO_SELECTION.USA;		// Regio selection, will affect to date/time formatting
	iLogger:				I_Logger := NullLogger();
END_VAR
VAR_OUTPUT
	
	oPersistencyHmi:		ST_PERSISTENCY_HMI;
END_VAR
VAR
	getHostName: 			FB_GetHostName;
	getAmsNetId:			FB_GetLocalAmsNetId;
	
	getLocalTime: 			FB_GetLocalTimeAndDate;
	
	blinkers:				FB_Blinkers;
	pulsers:				FB_Pulsers;
	
	
	persistency:			FB_Persistency;
	
	taskIndex:				DINT;		// The task index of the task in which we are called.
	
	pointerToByte:			POINTER TO BYTE;
END_VAR
VAR PERSISTENT
	numberOfPlcStarts:		UDINT;	// How often the PLC has been started
	timeOfPreviousCycle:	ULINT;
END_VAR

// Read epoch time
FC_CallAtStart_EpochTime();

// Read local system time as string
getLocalTime(iRegioSelection := iRegioSelection);

// Was used earlier to determine the cycleStart flag
IING.cycleTime := FC_GetEpochTime() - timeOfPreviousCycle;

// The famous cycle start flag, earlier done by checking the cycle time, TTECH-4497
taskIndex := GETCURTASKINDEXEX();	// -1 = The function is called from the Windows context.
									// 0 = The function is called from the real-time context, but not from a cyclic PLC task. This is the case, for example, with the automatic call of FB_init methods during initialization.
									// 1 to n = The function is called from a cyclic PLC task. The return value is the task index.
IF (taskIndex > 0) THEN
	IING.cycleStart :=  TwinCAT_SystemInfoVarList._TaskInfo[taskIndex].FirstCycle;
	IING.cycleCounter := TwinCAT_SystemInfoVarList._TaskInfo[taskIndex].CycleCount;
	IING.adsPort := TwinCAT_SystemInfoVarList._TaskInfo[taskIndex].AdsPort;
ELSE
	IING.cycleStart := FALSE;
	IING.cycleCounter := 0;
END_IF

IF (IING.cycleStart) THEN
	IncUDINT(numberOfPlcStarts);
	
	IING.pointerSize := SIZEOF(pointerToByte);
END_IF
timeOfPreviousCycle := FC_GetEpochTime();

// Read host name and AMS net id
getHostName(bExecute := IING.cycleStart, tTimeout := DEFAULT_ADS_TIMEOUT, sHostName => IING.localHostName);
getAmsNetId(bExecute := IING.cycleStart, tTimeOut := DEFAULT_ADS_TIMEOUT, AddrString => IING.localAmsNetId);


// Create blinking outputs
blinkers(oBlink100MS => IING.blink100MS, oBlink500MS => IING.blink500MS, oBlink1S => IING.blink1S, oBlink2S => IING.blink2S, oBlink5S => IING.blink5S,
	oBlink10S => IING.blink10S);
	
// Inverted blinks (good to make animations)
IING.invertedBlink100Ms := NOT IING.blink100MS;
IING.invertedBlink500Ms := NOT IING.blink500MS;
IING.invertedBlink1S := NOT IING.blink1S;
IING.invertedBlink2S := NOT IING.blink2S;
IING.invertedBlink5S := NOT IING.blink5S;
IING.invertedBlink10S := NOT IING.blink10S;
	
// Create periodic pulses
pulsers(oPulse100Ms => IING.pulse100Ms, oPulse500Ms => IING.pulse500Ms, oPulse1S => IING.pulse1S, oPulse2S => IING.pulse2S, oPulse10S => IING.pulse10S,
	oPulse30S => IING.pulse30S, oPulse1M => IING.pulse1M, oPulse1H => IING.pulse1H);





LOGGER.defaultLogger := iLogger;

{ IF defined(simulator) }
	IING.simulatorActive := TRUE;
{ ELSE }
	IING.simulatorActive := FALSE;
{ END_IF }

END_FUNCTION_BLOCK

// ---- LOGGING/NullLogger.TcPOU
FUNCTION NullLogger : I_Logger		// Returns a null logger instance

NullLogger := LOGGER.nullLogger;

END_FUNCTION

// ---- BASE/LocaleUtils/FB_GetLocalTimeAndDate.TcPOU
FUNCTION_BLOCK FB_GetLocalTimeAndDate	// Called from FB_Cyclestart, DO NOT call from your application 
										// Stores the local time/date to IIN.localTimeString/localDateString
										// Use FC_GetLocalTime and FC_GetLocalDate to retrieve those values
VAR_INPUT
	iRegioSelection:	E_REGIO_SELECTION;
END_VAR	
VAR_OUTPUT
	oCycleStart:		BOOL;			// Detection of a restart based on FB_LocalSystemTime
END_VAR
VAR
	year:				STRING(4);
	month: 				STRING(2);
	day: 				STRING(2);
	dayAsUint:			UINT;

	hour:				STRING(2);
	minute: 			STRING(2);
	second:				STRING(2);
	milliSecond:		STRING(3);
	
	dateString: 		STRING(10);
	timeString:	 		STRING(12);
	dateAndTimeString:	STRING(23);
	
	localSystemTime: 	FB_LocalSystemTime;
	
	previousDay:		UINT;
	localSystemTimeRtrig:	R_TRIG;
END_VAR

localSystemTime(bEnable := TRUE, dwCycle := 5, systemTime => IING.localSystemTime);

// It may take up to 5 PLC cycles before localSystemTime gives a valid time reading  
localSystemTimeRtrig(CLK := localSystemTime.bValid, Q => oCycleStart);

dayAsUint := WORD_TO_UINT(localSystemTime.systemTime.wDay);

day := FC_UintFormatter(iUint := dayAsUint, iLen := 2, iCharToPad := '0');
month := FC_UintFormatter(iUint := WORD_TO_UINT(localSystemTime.systemTime.wMonth), iLen := 2, iCharToPad := '0');
year := WORD_TO_STRING(localSystemTime.systemTime.wYear);

hour := FC_UintFormatter(iUint := WORD_TO_UINT(localSystemTime.systemTime.wHour), iLen := 2, iCharToPad := '0');
minute := FC_UintFormatter(iUint := WORD_TO_UINT(localSystemTime.systemTime.wMinute), iLen := 2, iCharToPad := '0');
second := FC_UintFormatter(iUint := WORD_TO_UINT(localSystemTime.systemTime.wSecond), iLen := 2, iCharToPad := '0');
milliSecond :=  FC_UintFormatter(iUint := WORD_TO_UINT(localSystemTime.systemTime.wMilliseconds), iLen := 3, iCharToPad := '0');
	

timeString := FC_2strConcatSeparator(iStr1 := hour, iStr2 := minute, iSeparator := IING.STRING_COLON);

// Short timestring for display in HMI
IING.localTimeMinAccuracy := FC_FormatTime(iRegioSelection := iRegioSelection, iHour := hour, iMinute := minute, iSeconds := IING.STRING_BLANK);

IING.localTimeSecAccuracy := FC_FormatTime(iRegioSelection := iRegioSelection, iHour := hour, iMinute := minute, iSeconds := second);

timeString := FC_2strConcatSeparator(iStr1 := timeString, iStr2 := second, iSeparator := IING.STRING_COLON);
timeString := FC_2strConcatSeparator(iStr1 := timeString, iStr2 := milliSecond, iSeparator := IING.STRING_COMMA); 

IING.usDateString := FC_3strConcatSeparator(iStr1 := year, iStr2 := month, iStr3:= day, iSeparator :=  IING.STRING_DASH);

CASE (iRegioSelection) OF
	E_REGIO_SELECTION.USA:
		dateString := IING.usDateString;
		
	E_REGIO_SELECTION.EUROPE:
		dateString := FC_3strConcatSeparator(iStr1 := day, iStr2 := month, iStr3:= year, iSeparator :=  IING.STRING_DASH);
END_CASE

IING.localDateString := dateString;
IING.localTimeString := timeString;
IING.localDateAndTimeString := FC_2strConcatSeparator(iStr1 := dateString, iStr2 := timeString, iSeparator := IING.STRING_SPACE);

IING.dayHasChanged := (dayAsUint <> previousDay);
previousDay := dayAsUint;

IING.iso8601Time := SYSTEMTIME_TO_ISO8601(systemTime := IING.localSystemTime, nBias := 0, bUTC := FALSE, nPrecision := 3);

END_FUNCTION_BLOCK

// ---- BASE/StringUtils/FC_UintFormatter.TcPOU
FUNCTION FC_UintFormatter : T_SHORT_STR	// UINT formatter (characters will be padded until desired string length is achieved)
VAR_INPUT
	iUint:			UINT;			// UINT to be formatted
	iLen:			UINT;			// Resulting formatted string length
	iCharToPad:		T_SHORT_STR;	// Character to be padded at the front
END_VAR
VAR
	uintStr:		T_SHORT_STR;
	strLen: 		UINT;
	charsToPad:		UINT;
	i:				UINT;	// for loop
END_VAR

uintStr := UINT_TO_STRING(iUint);
strLen := INT_TO_UINT(LEN(uintStr));

FC_UintFormatter := '';

charsToPad := iLen - strLen;

IF (charsToPad > 0) THEN
	FOR i := 0 TO (charsToPad - 1) DO
    	FC_UintFormatter := CONCAT(STR1 := FC_UintFormatter, STR2 := iCharToPad);
	END_FOR;
	FC_UintFormatter := CONCAT(STR1 := FC_UintFormatter, STR2 := uintStr);
ELSE
	FC_UintFormatter := uintStr;
END_IF;

END_FUNCTION

// ---- BASE/StringUtils/FC_2strConcatSeparator.TcPOU
FUNCTION FC_2strConcatSeparator : T_DEFAULT_STR	// Concatenates 2 strings with given separator
VAR_INPUT
	iSeparator:		STRING := IING.STRING_UNDERSCORE;	
	iStr1:			T_DEFAULT_STR;
	iStr2:			T_DEFAULT_STR;
END_VAR

FC_2strConcatSeparator := FC_3strConcat(iStr1 := iStr1, iStr2 := iSeparator, iStr3 := iStr2);

END_FUNCTION

// ---- BASE/StringUtils/FC_3strConcat.TcPOU
FUNCTION FC_3strConcat : T_DEFAULT_STR		// Concatenates 3 strings
VAR_INPUT
	iStr1:		T_DEFAULT_STR;
	iStr2:		T_DEFAULT_STR;
	iStr3:		T_DEFAULT_STR;
END_VAR

FC_3strConcat := CONCAT(CONCAT(iStr1, iStr2), iStr3);

END_FUNCTION

// ---- BASE/LocaleUtils/FC_FormatTime.TcPOU
FUNCTION FC_FormatTime : T_SHORT_STR	// Format the time according to regio selection
VAR_INPUT
	iRegioSelection:	E_REGIO_SELECTION;
	iHour:				STRING(2);
	iMinute:			STRING(2);
	iSeconds:			STRING(2);
END_VAR
VAR
	hour:				UINT;
	minute:				UINT;
	second:				UINT;
	pm:					BOOL := FALSE;
	
	secondsPassed:		bool;
END_VAR

hour := STRING_TO_UINT(iHour);
minute := STRING_TO_UINT(iMinute);

secondsPassed := FC_StringNotEmpty(iSeconds);
IF (secondsPassed) THEN
	second := STRING_TO_UINT(iSeconds);
END_IF

// Short version for display in HMI
CASE (iRegioSelection) OF
	E_REGIO_SELECTION.USA:
		IF (hour > 12) THEN
			pm := TRUE;
			hour := hour - 12;
		END_IF

		IF (secondsPassed) THEN
			FC_FormatTime := FC_3strConcatSeparator(iStr1 := FC_UintFormatter(iUint := hour, iLen := 2, iCharToPad := '0'),
				iStr2 := FC_UintFormatter(iUint := minute, iLen := 2, iCharToPad := '0'),
				iStr3 := FC_UintFormatter(iUint := second, iLen := 2, iCharToPad := '0'), iSeparator := IING.STRING_COLON);
		ELSE
			FC_FormatTime := FC_2strConcatSeparator(iStr1 := FC_UintFormatter(iUint := hour, iLen := 2, iCharToPad := '0'),
				iStr2 := FC_UintFormatter(iUint := minute, iLen := 2, iCharToPad := '0'), iSeparator := IING.STRING_COLON);
		END_IF

		IF (pm) THEN
			FC_FormatTime := FC_2strConcatSeparator(iStr1 := FC_FormatTime, iStr2 := IING.STRING_PM, iSeparator := IING.STRING_SPACE);
		ELSE
			FC_FormatTime := FC_2strConcatSeparator(iStr1 := FC_FormatTime, iStr2 := IING.STRING_AM, iSeparator := IING.STRING_SPACE);
		END_IF
	
	E_REGIO_SELECTION.EUROPE:
		IF (secondsPassed) THEN
			FC_FormatTime := FC_3strConcatSeparator(iStr1 := FC_UintFormatter(iUint := hour, iLen := 2, iCharToPad := '0'),
				iStr2 := FC_UintFormatter(iUint := minute, iLen := 2, iCharToPad := '0'),
				iStr3 := FC_UintFormatter(iUint := second, iLen := 2, iCharToPad := '0'), iSeparator := IING.STRING_COLON);
		ELSE
			FC_FormatTime := FC_2strConcatSeparator(iStr1 := FC_UintFormatter(iUint := hour, iLen := 2, iCharToPad := '0'),
				iStr2 := FC_UintFormatter(iUint := minute, iLen := 2, iCharToPad := '0'), iSeparator := IING.STRING_COLON);
		END_IF
END_CASE

END_FUNCTION

// ---- BASE/StringUtils/FC_StringNotEmpty.TcPOU
FUNCTION FC_StringNotEmpty : BOOL
VAR_INPUT
	iString:	T_DEFAULT_STR;
END_VAR

FC_StringNotEmpty := LEN(iString) > 0;

END_FUNCTION

// ---- BASE/StringUtils/FC_3strConcatSeparator.TcPOU
FUNCTION FC_3strConcatSeparator : T_DEFAULT_STR		// Concatenates 3 strings with given separator
VAR_INPUT
	iSeparator:		STRING := IING.STRING_UNDERSCORE;
	iStr1:			T_DEFAULT_STR;
	iStr2:			T_DEFAULT_STR;
	iStr3:			T_DEFAULT_STR;
END_VAR

FC_3strConcatSeparator := FC_2strConcatSeparator(iSeparator := iSeparator,
	iStr1 := FC_2strConcatSeparator(iSeparator := iSeparator, iStr1 := iStr1, iStr2 := iStr2), iStr2 := iStr3);

END_FUNCTION

// ---- BASE/PulsersBlinkers/FB_Blinkers.TcPOU
FUNCTION_BLOCK FB_Blinkers		// Called from FB_Cyclestart, DO NOT call from your application
								// Collection of blinkers
VAR_OUTPUT
	oBlink100Ms: 	BOOL;
	oBlink500Ms: 	BOOL;
	oBlink1S: 		BOOL;
	oBlink2S:		BOOL;
	oBlink5S:		BOOL;
	oBlink10S: 		BOOL;
END_VAR
VAR
	blink100Ms:		FB_Blink;
	blink500Ms: 	FB_Blink;
	blink1S:		FB_Blink;
	blink2S:		FB_Blink;
	blink5S:		FB_Blink;
	blink10S:		FB_Blink;
END_VAR

blink100Ms(iTime := T#100MS, oBlink => oBlink100Ms);
blink500Ms(iTime := T#500MS, oBlink => oBlink500Ms);
blink1S(iTime := T#1S, oBlink => oBlink1S);
blink2S(iTime := T#2S, oBlink => oBlink2S);
blink5S(iTime := T#5S, oBlink => oBlink5S);
blink10S(iTime := T#10S, oBlink => oBlink10S);

END_FUNCTION_BLOCK

// ---- BASE/PulsersBlinkers/FB_Blink.TcPOU
FUNCTION_BLOCK FB_Blink		// Blink at the specified time
VAR_INPUT
	iTime:		TIME;		// Blinking time
END_VAR
VAR_OUTPUT
	oBlink:		BOOL;		// The blinker (iTime TRUE followed by iTime FALSE)
END_VAR
VAR
	ton:		TON;
	tof: 		TOF;
END_VAR

ton(IN := NOT (oBlink), PT := iTime);
tof(IN := ton.Q, PT := iTime, Q => oBlink);

END_FUNCTION_BLOCK

// ---- BASE/PulsersBlinkers/FB_Pulsers.TcPOU
FUNCTION_BLOCK FB_Pulsers		// Called from FB_Cyclestart, DO NOT call from your application
								// Collection of pulsers

VAR_OUTPUT
	oPulse100Ms:		BOOL;
	oPulse500Ms:		BOOL;
	oPulse1S:			BOOL;
	oPulse2S:			BOOL;
	oPulse10S:			BOOL;
	oPulse30S:			BOOL;
	oPulse1M:			BOOL;
	oPulse1H:			BOOL;
END_VAR
VAR
	pulse100Ms:			FB_Pulse;
	pulse500Ms:			FB_Pulse;
	pulse1S:			FB_Pulse;
	pulse2S:			FB_Pulse;
	pulse10S:			FB_Pulse;
	pulse30S:			FB_Pulse;
	pulse1M:			FB_Pulse;
	pulse1H:			FB_Pulse;
END_VAR

pulse100Ms(iTime := T#100MS, oPulse => oPulse100Ms);
pulse500Ms(iTime := T#500MS, oPulse => oPulse500Ms);
pulse1S(iTime := T#1S, oPulse => oPulse1S);
pulse2S(iTime := T#2S, oPulse => oPulse2S);
pulse10S(iTime := T#10S, oPulse => oPulse10S);
pulse30S(iTime := T#30S, oPulse => oPulse30S);
pulse1M(iTime := T#1M, oPulse => oPulse1M);
pulse1H(iTime := T#1H, oPulse => oPulse1H);

END_FUNCTION_BLOCK

// ---- BASE/PulsersBlinkers/FB_Pulse.TcPOU
FUNCTION_BLOCK FB_Pulse			// Pulse (= 1 plc cycle) at the specified time
VAR_INPUT
	iTime:		TIME;			// Pulsing time
END_VAR
VAR_OUTPUT
	oPulse:		BOOL;			// The pulser (iTime FALSE followed by a 1 plc cycle TRUE)
END_VAR
VAR
	pulse:		TON;
END_VAR

pulse(IN := TRUE, PT := iTime);
oPulse := pulse.Q;
IF (pulse.Q) THEN
	pulse(IN := FALSE);
END_IF

END_FUNCTION_BLOCK

// ---- BASE/Persistency/FB_Persistency.TcPOU
FUNCTION_BLOCK FB_Persistency		// Called from FB_Cyclestart, DO NOT call from your application
VAR_INPUT
	iExtSave:					BOOL;	// An external sav e trigger (eg. from a UPS function)
END_VAR
VAR_OUTPUT
	oOut:						ST_PERSISTENCY_OUT;
	oHmi:						ST_PERSISTENCY_HMI;
END_VAR
VAR
	pulser:						FB_Pulse;
	extSaveEdge:				R_TRIG;
	saveNowEdge:				R_TRIG;
	doSave:						BOOL;
	write:						FB_WritePersistentData;
	service:					ST_PERSISTENCY_SERVICE;
END_VAR
VAR PERSISTENT	
	settings:					ST_PERSISTENCY_SETTINGS;
END_VAR

pulser(iTime := settings.saveInterval);

extSaveEdge(CLK := iExtSave);
saveNowEdge(CLK := service.saveNow);


doSave := saveNowEdge.Q OR extSaveEdge.Q OR (settings.autoSave AND pulser.oPulse);

write(PORT := settings.port, START := doSave, TMOUT := T#2S, MODE := E_PersistentMode.SPDM_VAR_BOOST,
	BUSY => oOut.busy, ERR => oOut.error, ERRID => oOut.beckhoffErrorId);
	
oOut.errorIdEnum := FC_GetAdsErrorCode(oOut.beckhoffErrorId);

hmi();

METHOD PRIVATE hmi : BOOL

oHmi.service REF= service;
oHmi.settings REF= settings;
oHmi.out REF= oOut;
END_METHOD

END_FUNCTION_BLOCK

// ---- BASE/AdsUtils/FC_GetAdsErrorCode.TcPOU
FUNCTION FC_GetAdsErrorCode : E_ADS_ERRORS		// Converts an error number into an ADS enum error code
VAR_INPUT
	iErrorCode:	UDINT;		// The error code as a number
END_VAR

CASE iErrorCode OF
	0:
		FC_GetAdsErrorCode := E_ADS_ERRORS.NO_ERROR;

	6:
		FC_GetAdsErrorCode := E_ADS_ERRORS.TARGET_PORT_NOT_FOUND;
		
	7:
		FC_GetAdsErrorCode := E_ADS_ERRORS.TARGET_MACHINE_NOT_FOUND;
	
	1792:
		FC_GetAdsErrorCode := E_ADS_ERRORS.ADSERR_DEVICE_ERROR;
	
	1793:
		FC_GetAdsErrorCode := E_ADS_ERRORS.ADSERR_DEVICE_SRVNOTSUPP; 
	
	1794:
		FC_GetAdsErrorCode := E_ADS_ERRORS.ADSERR_DEVICE_INVALIDGRP; 
	
	1795:
		FC_GetAdsErrorCode := E_ADS_ERRORS.ADSERR_DEVICE_INVALIDOFFSET;
	
	1796:
		FC_GetAdsErrorCode := E_ADS_ERRORS.ADSERR_DEVICE_INVALIDACCESS;
	
	1797:
		FC_GetAdsErrorCode := E_ADS_ERRORS.ADSERR_DEVICE_INVALIDSIZE;

	1798:
		FC_GetAdsErrorCode := E_ADS_ERRORS.ADSERR_DEVICE_INVALIDDATA;

	1799:
		FC_GetAdsErrorCode := E_ADS_ERRORS.ADSERR_DEVICE_NOTREADY;

	1800:
		FC_GetAdsErrorCode := E_ADS_ERRORS.ADSERR_DEVICE_BUSY;

	1801:
		FC_GetAdsErrorCode := E_ADS_ERRORS.ADSERR_DEVICE_INVALIDCONTEXT;

	1802:
		FC_GetAdsErrorCode := E_ADS_ERRORS.ADSERR_DEVICE_NOMEMORY;
	
	1803:
		FC_GetAdsErrorCode := E_ADS_ERRORS.ADSERR_DEVICE_INVALIDPARM;
	
	1804:
		FC_GetAdsErrorCode := E_ADS_ERRORS.ADSERR_DEVICE_NOTFOUND;		// Eg. Opening a file which does not exist
	
	1805:
		FC_GetAdsErrorCode := E_ADS_ERRORS.ADSERR_DEVICE_SYNTAX;
	
	1806:
		FC_GetAdsErrorCode := E_ADS_ERRORS.ADSERR_DEVICE_INCOMPATIBLE;
	
	1807:
		FC_GetAdsErrorCode := E_ADS_ERRORS.ADSERR_DEVICE_EXISTS;
	
	1808:
		FC_GetAdsErrorCode := E_ADS_ERRORS.ADSERR_DEVICE_SYMBOLNOTFOUND;
	
	1809:
		FC_GetAdsErrorCode := E_ADS_ERRORS.ADSERR_DEVICE_SYMBOLVERSIONINVAL;
	
	1810:
		FC_GetAdsErrorCode := E_ADS_ERRORS.ADSERR_DEVICE_INVALIDSTATE;

	1811:
		FC_GetAdsErrorCode := E_ADS_ERRORS.ADSERR_DEVICE_TRANSMODENOTSUPP;
	
	1812:
		FC_GetAdsErrorCode := E_ADS_ERRORS.ADSERR_DEVICE_NOTIFYHNDINVALID;
	
	1813:
		FC_GetAdsErrorCode := E_ADS_ERRORS.ADSERR_DEVICE_CLIENTUNKNOWN;
	
	1814:
		FC_GetAdsErrorCode := E_ADS_ERRORS.ADSERR_DEVICE_NOMOREHDLS;
	
	1815:
		FC_GetAdsErrorCode := E_ADS_ERRORS.ADSERR_DEVICE_INVALIDWATCHSIZE;
	
	1816:
		FC_GetAdsErrorCode := E_ADS_ERRORS.ADSERR_DEVICE_NOTINIT;
	
	1817:
		FC_GetAdsErrorCode := E_ADS_ERRORS.ADSERR_DEVICE_TIMEOUT;
	
	1818:
		FC_GetAdsErrorCode := E_ADS_ERRORS.ADSERR_DEVICE_NOINTERFACE;
	
	1819:
		FC_GetAdsErrorCode := E_ADS_ERRORS.ADSERR_DEVICE_INVALIDINTERFACE;
	
	1820:
		FC_GetAdsErrorCode := E_ADS_ERRORS.ADSERR_DEVICE_INVALIDCLSID;
	
	1821:
		FC_GetAdsErrorCode := E_ADS_ERRORS.ADSERR_DEVICE_INVALIDOBJID;
	
	1822:
		FC_GetAdsErrorCode := E_ADS_ERRORS.ADSERR_DEVICE_PENDING;
	
	1823:
		FC_GetAdsErrorCode := E_ADS_ERRORS.ADSERR_DEVICE_ABORTED;
	
	1824:
		FC_GetAdsErrorCode := E_ADS_ERRORS.ADSERR_DEVICE_WARNING;
	
	1825:
		FC_GetAdsErrorCode := E_ADS_ERRORS.ADSERR_DEVICE_INVALIDARRAYIDX;
	
	1826:
		FC_GetAdsErrorCode := E_ADS_ERRORS.ADSERR_DEVICE_SYMBOLNOTACTIVE;
	
	1827:
		FC_GetAdsErrorCode := E_ADS_ERRORS.ADSERR_DEVICE_ACCESSDENIED;
	
	1828:
		FC_GetAdsErrorCode := E_ADS_ERRORS.ADSERR_DEVICE_LICENSENOTFOUND;
	
	1829:
		FC_GetAdsErrorCode := E_ADS_ERRORS.ADSERR_DEVICE_LICENSEEXPIRED;
	
	1830:
		FC_GetAdsErrorCode := E_ADS_ERRORS.ADSERR_DEVICE_LICENSEEXCEEDED;
	
	1831:
		FC_GetAdsErrorCode := E_ADS_ERRORS.ADSERR_DEVICE_LICENSEINVALID;
	
	1832:
		FC_GetAdsErrorCode := E_ADS_ERRORS.ADSERR_DEVICE_LICENSESYSTEMID;
	
	1833:
		FC_GetAdsErrorCode := E_ADS_ERRORS.ADSERR_DEVICE_LICENSENOTIMELIMIT;
	
	1834:
		FC_GetAdsErrorCode := E_ADS_ERRORS.ADSERR_DEVICE_LICENSEFUTUREISSUE;
	
	1835:
		FC_GetAdsErrorCode := E_ADS_ERRORS.ADSERR_DEVICE_LICENSETIMETOLONG;
	
	1836:
		FC_GetAdsErrorCode := E_ADS_ERRORS.ADSERR_DEVICE_EXCEPTION;
	
	1837:
		FC_GetAdsErrorCode := E_ADS_ERRORS.ADSERR_DEVICE_LICENSEDUPLICATED;
	
	1838:
		FC_GetAdsErrorCode := E_ADS_ERRORS.ADSERR_DEVICE_SIGNATUREINVALID;
	
	1839:
		FC_GetAdsErrorCode := E_ADS_ERRORS.ADSERR_DEVICE_CERTIFICATEINVALID;
	
	1856:
		FC_GetAdsErrorCode := E_ADS_ERRORS.ADSERR_CLIENT_ERROR;
	
	1857:
		FC_GetAdsErrorCode := E_ADS_ERRORS.ADSERR_CLIENT_INVALIDPARM;

	1858:
		FC_GetAdsErrorCode := E_ADS_ERRORS.ADSERR_CLIENT_LISTEMPTY;

	1859:
		FC_GetAdsErrorCode := E_ADS_ERRORS.ADSERR_CLIENT_VARUSED;

	1860:
		FC_GetAdsErrorCode := E_ADS_ERRORS.ADSERR_CLIENT_DUPLINVOKEID;

	1861:
		FC_GetAdsErrorCode := E_ADS_ERRORS.ADSERR_CLIENT_SYNCTIMEOUT;

	1862:
		FC_GetAdsErrorCode := E_ADS_ERRORS.ADSERR_CLIENT_W32ERROR;

	1863:
		FC_GetAdsErrorCode := E_ADS_ERRORS.ADSERR_CLIENT_TIMEOUTINVALID;

	1864:
		FC_GetAdsErrorCode := E_ADS_ERRORS.ADSERR_CLIENT_PORTNOTOPEN;

	1872:
		FC_GetAdsErrorCode := E_ADS_ERRORS.ADSERR_CLIENT_NOAMSADDR;

	1873:
		FC_GetAdsErrorCode := E_ADS_ERRORS.ADSERR_CLIENT_SYNCINTERNAL;

	1874:
		FC_GetAdsErrorCode := E_ADS_ERRORS.ADSERR_CLIENT_ADDHASH;

	1875:
		FC_GetAdsErrorCode := E_ADS_ERRORS.ADSERR_CLIENT_REMOVEHASH;

	1876:
		FC_GetAdsErrorCode := E_ADS_ERRORS.ADSERR_CLIENT_NOMORESYM;

	1877:
		FC_GetAdsErrorCode := E_ADS_ERRORS.ADSERR_CLIENT_SYNCRESINVALID;

	ELSE
		FC_GetAdsErrorCode := E_ADS_ERRORS.TODO;
	
END_CASE

END_FUNCTION

// ---- BASE/LocaleUtils/FC_CallAtStart_EpochTime.TcPOU
FUNCTION FC_CallAtStart_EpochTime : BOOL		// Called from FB_Cyclestart, DO NOT call from your application
												// Stores the EPOCH time to IIN.epochtime

// To be called once/cycle

IING.epochtime := (F_GetSystemTime() / 10000) - IING.EPOCH_CORRECTION;	// System is in 100nseconds -> divide by 10000 for milliseconds

END_FUNCTION

// ---- BASE/LocaleUtils/FC_GetEpochTime.TcPOU
FUNCTION FC_GetEpochTime : ULINT	// Returns the current EPOCH time

FC_GetEpochTime := IING.epochtime;

END_FUNCTION

// ---- BASE/NumberUtils/IncUDINT.TcPOU
FUNCTION IncUDINT : UDINT		// Increments the given UINT value
VAR_IN_OUT
	ioNum:	UDINT;		// Value to increment
END_VAR

IncUDINT := ioNum := ioNum + 1;

END_FUNCTION

// ---- DATA/REPORTING/FB_DummyDataReporter.TcPOU
FUNCTION_BLOCK FB_DummyDataReporter IMPLEMENTS I_DataReporter		// Dummy data reporter
	// This will be returned to the caller if no real implementation is found.
	// Methods in this FB will do nothing, thus the project can run happily

METHOD PUBLIC ic_deviceSpeedChanged	// To be called when the (device) speed changes
VAR_INPUT
	iPos:			E_POS;				// Position enumerate
	iMiscArea:		T_SHORT_STR;		// Safety or misc area enumerate (string). If defined/non-empty, use this instead of iPos
	iNew:			INT;				// The new speed value
END_VAR
END_METHOD

METHOD PUBLIC ic_initializeDone	// To be called when a initialization (aka hard reset) is done
VAR_INPUT
	iPos:			E_POS;				// The position
	iMiscArea:		T_SHORT_STR;		// Safety or misc area enumerate (string). If defined/non-empty, use this instead of iPos
	iOrigin:		E_RESET_ORIGIN;
END_VAR
END_METHOD

METHOD PUBLIC ic_operationModeChanged	// To be called when the control signal operation mode changes
VAR_INPUT
	iPos:			E_POS;				// The position
	iMiscArea:		T_SHORT_STR;		// Safety or misc area enumerate (string). If defined/non-empty, use this instead of iPos
	iNew:			E_OPERATION_MODE;	// New operation mode
END_VAR
END_METHOD

METHOD PUBLIC ic_resetDone	// To be called when a reset is done
VAR_INPUT
	iPos:			E_POS;				// The position
	iMiscArea:		T_SHORT_STR;		// Safety or misc area enumerate (string). If defined/non-empty, use this instead of iPos
	iOrigin:		E_RESET_ORIGIN;
	iResetKeyLabel:	T_SHORT_STR;		// What reset key was pressed
END_VAR
END_METHOD

METHOD PUBLIC ic_serviceStateChanged		// To be called when the (control signal) service state changes
VAR_INPUT
	iPos:			E_POS;				// The position
	iMiscArea:		T_SHORT_STR;		// Safety or misc area enumerate (string). If defined/non-empty, use this instead of iPos
	iState:			BOOL;				// TRUE = service activated, FALSE = service deactivated
END_VAR
END_METHOD

END_FUNCTION_BLOCK

// ---- LOGGING/NullLogger/FB_NullLogger.TcPOU
FUNCTION_BLOCK FB_NullLogger IMPLEMENTS I_Logger				// Null logger implementation

METHOD PUBLIC debug : BOOL	// Logs the data with log level 'DEBUG'
VAR_INPUT
	iData:		T_DEFAULT_STR;						// Data to be logged, limited to 255 characters
END_VAR
// Do nothing
END_METHOD

METHOD PUBLIC deregister : BOOL
VAR_INPUT
	iWho:				T_SHORT_STR;
END_VAR
END_METHOD

METHOD PUBLIC doLog : BOOL
VAR_INPUT
	iData:		T_DEFAULT_STR;						// Data to be logged, limited to 255 characters
	iLevel:		E_LOG_LEVEL := E_LOG_LEVEL.ERROR;	// Log level
END_VAR
END_METHOD

METHOD PUBLIC error : BOOL	// Logs the data with log level 'ERROR'
VAR_INPUT
	iData:		T_DEFAULT_STR;						// Data to be logged, limited to 255 characters
END_VAR
// Do nothing
END_METHOD

METHOD PUBLIC info : BOOL	// Logs the data with log level 'INFO'
VAR_INPUT
	iData:		T_DEFAULT_STR;						// Data to be logged, limited to 255 characters
END_VAR
// Do nothing
END_METHOD

METHOD PUBLIC register : BOOL
VAR_INPUT
	iWho:		T_SHORT_STR;
	iObserver:	I_Logger;
END_VAR
END_METHOD

METHOD PUBLIC trace : BOOL	// Logs the data with log level 'TRACE'
VAR_INPUT
	iData:		T_DEFAULT_STR;						// Data to be logged, limited to 255 characters
END_VAR
// Do nothing
END_METHOD

METHOD PUBLIC warn : BOOL	// Logs the data with log level 'WARN'
VAR_INPUT
	iData:		T_DEFAULT_STR;						// Data to be logged, limited to 255 characters
END_VAR
// Do nothing
END_METHOD

END_FUNCTION_BLOCK

// ---- ALARMS/AppSupport/FB_Interceptor.TcPOU
FUNCTION_BLOCK FB_Interceptor
VAR_INPUT
	iDebugEnableBreakpoint:	BOOL;			// When TRUE, stepping will stop as long as the debugging is ON
END_VAR
VAR_IN_OUT
	ioDebugAllowSingleStep:	BOOL;			// When TRUE, a single step will be allowed, then the debugger becomes active again
END_VAR
VAR
	interceptors:	ARRAY[0..3] OF ST_INTERCEPTOR;
	cnt:			INT;
END_VAR

METHOD PUBLIC getResult : ST_INTERCEPTOR_RESULT
VAR
	i:	INT;
END_VAR
{warning disable C0371}

getResult.clear := TRUE;
getResult.missing := IING.STRING_BLANK;

IF (cnt > 0) THEN
	FOR i := 0 TO cnt - 1 DO
		IF (NOT interceptors[i].check) THEN
			getResult.clear := FALSE;						// This interceptor check fails
			getResult.missing := interceptors[i].desc;		// Set the reason why this interceptor failed
			RETURN;
		END_IF
	END_FOR
END_IF

// We come here when all interceptors were good
IF (iDebugEnableBreakpoint) THEN
	IF (ioDebugAllowSingleStep) THEN
		ioDebugAllowSingleStep := FALSE;
	ELSE
		getResult.clear := FALSE;							// We stop program continuation by taking the 'clear' flag off 
		getResult.missing := 'DEBUG';						// We tell to the user that the debugger is active
	END_IF
END_IF

{warning restore C0371}
END_METHOD

METHOD public init : BOOL
cnt := 0;

// Just in case
interceptors[0].check := TRUE;
interceptors[0].desc := 'this interceptor is not in use';

interceptors[1].check := TRUE;
interceptors[1].desc := 'this interceptor is not in use';

interceptors[2].check := TRUE;
interceptors[2].desc := 'this interceptor is not in use';
END_METHOD

METHOD PUBLIC set1Interceptor : BOOL
VAR_INPUT
	check1:	BOOL;
	desc1:	T_SHORT_STR;
END_VAR
interceptors[0].check := check1;
interceptors[0].desc := desc1;
cnt := 1;

// Just in case
interceptors[1].check := TRUE;
interceptors[1].desc := 'this interceptor is not in use';

interceptors[2].check := TRUE;
interceptors[2].desc := 'this interceptor is not in use';
END_METHOD

METHOD PUBLIC set2Interceptor : BOOL
VAR_INPUT
	check1:		BOOL;
	desc1:		T_SHORT_STR;
	check2:		BOOL;
	desc2:		T_SHORT_STR;
END_VAR
interceptors[0].check := check1;
interceptors[0].desc := desc1;
interceptors[1].check := check2;
interceptors[1].desc := desc2;
cnt := 2;

// Just in case
interceptors[2].check := TRUE;
interceptors[2].desc := 'this interceptor is not in use';
END_METHOD

METHOD PUBLIC set3Interceptor : BOOL
VAR_INPUT
	check1:		BOOL;
	desc1:		T_SHORT_STR;
	check2:		BOOL;
	desc2:		T_SHORT_STR;
	check3:		BOOL;
	desc3:		T_SHORT_STR;
END_VAR
interceptors[0].check := check1;
interceptors[0].desc := desc1;
interceptors[1].check := check2;
interceptors[1].desc := desc2;
interceptors[2].check := check3;
interceptors[2].desc := desc3;
cnt := 3;
END_METHOD

METHOD PUBLIC set4Interceptor : BOOL
VAR_INPUT
	iCheck1:	BOOL;
	iDesc1:		T_SHORT_STR;
	iCheck2:	BOOL;
	iDesc2:		T_SHORT_STR;
	iCheck3:	BOOL;
	iDesc3:		T_SHORT_STR;
	iCheck4:	BOOL;
	iDesc4:		T_SHORT_STR;
END_VAR
interceptors[0].check := iCheck1;
interceptors[0].desc := iDesc1;
interceptors[1].check := iCheck2;
interceptors[1].desc := iDesc2;
interceptors[2].check := iCheck3;
interceptors[2].desc := iDesc3;
interceptors[3].check := iCheck4;
interceptors[3].desc := iDesc4;
cnt := 4;
END_METHOD

END_FUNCTION_BLOCK

// ---- ALARMS/AppSupport/FB_StepperProgram.TcPOU
{attribute 'reflection'} 
FUNCTION_BLOCK FB_StepperProgram EXTENDS FB_BaseWithAlarmEvents  	// Base skeleton for a stepping program
VAR
	stepChanged:				BOOL;				// TRUE when step change has happened
	interceptor:				FB_Interceptor;
	conditionCacheActive:		BOOL;				// When TRUE, condition caching is activated (so 1 PLC cycle iCondition pulses dont get lost)
	conditionCache:				BOOL;				// Help var that caches the iCondition (TRUE) signal when paused or interceptor is 'active'
	stepPtr:					POINTER TO INT;		// Needed for casting the step (as INT) back to step (as ENUM)
	
	enableDebug:				BOOL;				// Set TRUE to activate debugging (stepping will stop)
	maxDebugTon:				TON; 
	debugAllowSingleStep:		BOOL;				// When TRUE, a single step will be allowed, THEN the debugger becomes active again
	
	stepDuration:				TIME;				// The time/duration we have been in the current step
	
    {attribute 'instance-path'} 
    {attribute 'noinit'} 
	instancePath:				T_SHORT_STR;
	
	stoppedBoolLogger:			FB_BoolLogger;
	stopped2BoolLogger:			FB_BoolLogger;
	
	pauseInNextCycle:			BOOL;				// Used by pauseAsNeededWithOneCycleDelay
	
	interceptorFailed:			BOOL;				// If interceptor fails in condition x, it will also fail in condition y
	
	manualBehaviorIsSameAsPause:	BOOL;
	
	// Helpers
	hardResetPulseForStepperProgram:	BOOL;
	hardResetPulseDueToGlobalReset:		BOOL;		// helper flag when global reset is called (= a method)
END_VAR
VAR PERSISTENT
	oldStepForStepChangeOnly:	INT;
	prevStep:					INT;
	maxDebugTime:				TIME := T#1M;		// The debugger will stay active for a maximum of this time (so not staying ON forever)
	stepStartedTime:			TIME;				// For calculating time duration of the current step
END_VAR
VAR_OUTPUT
	oDebugStep:					T_SHORT_STR;		// For showing the STEP in Engineering VISU
	oUserInfo:					T_SHORT_STR;
	oStopped:					BOOL;				// TRUE when the sequence is halted due to manual mode or pause request
END_VAR

METHOD PROTECTED callMeRightAfterSwitchCase : BOOL	// MUST to be called after the SWITCH CASE, otherwise the stepChanged is set too late
VAR_INPUT
	iLogTraces:		BOOL := TRUE;
	iExtraTrace:	T_SHORT_STR;
END_VAR
VAR
//	areas:			ST_GLOBAL_RESET_AREAS;
	primaryArea:	INT;
	secondaryArea:	INT;
END_VAR
updateOldStep();
trace(iLogTraces, iExtraTrace);

hardResetPulseForStepperProgram := FALSE;
IF (iControlSignalsIf <> IING.ZERO_POINTER) THEN
	// Keep iControlSignals here for now (conveyor overwrites it)
	hardResetPulseForStepperProgram := iControlSignals.hardResetPulse OR iControlSignalsIf.ic_getControlSignalsOutPtr()^.hardResetPulse; 
ELSE
	hardResetPulseForStepperProgram := iControlSignals.hardResetPulse;
END_IF

hardResetPulseForStepperProgram := hardResetPulseForStepperProgram OR hardResetPulseDueToGlobalReset; 
hardResetPulseDueToGlobalReset := FALSE;

IF (hardResetPulseForStepperProgram) THEN
	conditionCache := FALSE;			// After hard reset, the iCondition TRUE cache must always be cleared
	initDebugger();
	interceptor.init();
	hardResetWasCalled();				// Here project specific stuff is to be implemented
END_IF

// Setting this event based causes steps not being visible after hard reset, lets keep it updating this way  
IF (IING.pulse100Ms) THEN
	oDebugStep := stepAsString();
END_IF
	
maxDebugTon(IN := enableDebug, PT := maxDebugTime);
IF (maxDebugTon.Q) THEN
	initDebugger();
END_IF

stoppedBoolLogger(iIn := oStopped, iLogRising := TRUE, iLogFalling := TRUE,  iPos := iPos, iDeviceType := iDeviceType, iDeviceId := 'oHalted');
mHandleSubPausing();
stopped2BoolLogger(iIn := oStopped, iLogRising := TRUE, iLogFalling := TRUE,  iPos := iPos, iDeviceType := iDeviceType, iDeviceId := 'oHalted again');


// we have passed all gotoNextStep's, reset this flag
interceptorFailed := FALSE;
END_METHOD

METHOD PROTECTED callMeRightBeforeSwitchCase : BOOL	// MUST be called before the SWITCH CASE
VAR_INPUT
	iStepPtr:	POINTER TO INT;		// Pointer to your ENUM step
END_VAR
stepPtr := iStepPtr;
oStopped := FALSE;
conditionCacheActive := FALSE;	// Need to be activated in each PLC cycle

interceptor(iDebugEnableBreakpoint := enableDebug, ioDebugAllowSingleStep := debugAllowSingleStep);

stepDuration := (TIME() - stepStartedTime);
END_METHOD

METHOD PROTECTED enableConditionCache : BOOL		// Enables caching of iCondition in gotoNextStep
conditionCacheActive := TRUE;
END_METHOD

METHOD PROTECTED gotoNextStep : BOOL	// To be called from gotoNextStep
VAR_INPUT
	iCondition:			BOOL;	// When TRUE, your stepping program will goto iNextStep
	iNextStep:			INT;	// Nextstep (as INT), conversion to INT happens automatically
END_VAR
VAR
	interceptorResult:	ST_INTERCEPTOR_RESULT;
END_VAR
IF (NOT (stepPtr^ <> oldStepForStepChangeOnly) AND NOT interceptorFailed) THEN
	IF (oStopped) THEN
		oUserInfo := 'Paused';
		setConditionCache(iCondition, 'Condition cached from pause, current step: ');
	ELSE
		IF (iCondition OR (conditionCacheActive AND conditionCache)) THEN
			interceptorResult := interceptor.getResult();
			IF (interceptorResult.clear) THEN
				IF (NOT iCondition) THEN	// If we get here, it is coming through a cached condition
					FC_GetLogger().info(iData := FC_3strConcat(iStr1:= getLoggingId(), iStr2 := ', ', iStr3 := 'Cached condition caused step change'));
				END_IF
			
				// We are good to proceed to the next step
				stepPtr^ := iNextStep;			// We write the step variable here
				conditionCache := FALSE;		// Reset the iCondition cache
	
				oUserInfo := IING.STRING_BLANK;
				
				pauseInNextCycle := FALSE;		// If pause didnt happen, this need to be reset again
			ELSE
				oUserInfo := interceptorResult.missing;					
				setConditionCache(iCondition, 'Condition cached from interceptor, current step: ');
				
				interceptorFailed := TRUE;
			END_IF
		ELSE	// No pausing, nothing we are waiting for -> clear the UserInfo
			oUserInfo := IING.STRING_BLANK;
		END_IF
	END_IF
END_IF
END_METHOD

METHOD PROTECTED hardResetWasCalled : BOOL		// Can be used to execute 'hard reset' functionality, overwrite in your implementation
// Overwrite in your stepping program implementation
END_METHOD

METHOD PUBLIC ic_getCurrentStep : T_SHORT_STR		// Returns the current step of this FB -> for visualization purposes
ic_getCurrentStep := stepAsString();
END_METHOD

METHOD PUBLIC ic_getName : T_SHORT_STR		// Return the instance name of this FB
ic_getName := instancePath;
END_METHOD

METHOD PUBLIC ic_isInAuto : BOOL		// Return TRUE when in AUTO
IF (iControlSignalsIf <> IING.ZERO_POINTER) THEN
	ic_isInAuto := iControlSignalsIf.ic_isInAuto();
ELSE
	ic_isInAuto := iControlSignals.auto;
END_IF
END_METHOD

METHOD PUBLIC ic_isPauseByCsRequested : BOOL		// Is Pause by control signals requested
IF (iControlSignalsIf <> IING.ZERO_POINTER) THEN
	ic_isPauseByCsRequested := iControlSignalsIf.ic_isInPause();
ELSE
	ic_isPauseByCsRequested := iControlSignals.pauseRequest;
END_IF
END_METHOD

METHOD PUBLIC ic_isReady : BOOL			// Return TRUE when this sequence is READY to start over
ic_isReady := FALSE;
END_METHOD

METHOD public ic_isSaOk : BOOL		// // Return TRUE when this safety area is ok
ic_isSaOk := FALSE;
END_METHOD

METHOD PUBLIC ic_putToAutoAndUnpause		// Called by FB_GlobalResetArea when sequence is to switch to AUTO and NOT PAUSE
IF (iControlSignalsIf <> IING.ZERO_POINTER) THEN
	iControlSignalsIf.ic_switchToAuto();
	iControlSignalsIf.ic_unPause();
END_IF
END_METHOD

METHOD PRIVATE initDebugger : BOOL
enableDebug := FALSE;
debugAllowSingleStep := FALSE;
END_METHOD

METHOD PUBLIC isTimeExpired : BOOL		// Returns TRUE when the given time is bigger than the current step duration  
VAR_INPUT
	iTime:	TIME;
END_VAR
isTimeExpired := (stepDuration >= iTime);
END_METHOD

METHOD PROTECTED mHandleSubPausing		// Here you can overwrite the oStopped with information from your sub sequences
// Overwrite in your stepping program implementation
// oStoppped := oStopped and mySubSequence.oStopped;
END_METHOD

METHOD PROTECTED mIsManualBehaviorSameAsPause :	BOOL	// Return TRUE when going to Manual is to behave same as Pause
														// Overwrite as needed in your sequence
mIsManualBehaviorSameAsPause := FALSE;
END_METHOD

METHOD PROTECTED mIsPauseByManualRequested : BOOL		// TRUE means we request pause (because we are in manual)
														// Not intended to be overriden in your application
mIsPauseByManualRequested := mIsManualBehaviorSameAsPause() AND NOT ic_isInAuto();
END_METHOD

METHOD PROTECTED mPurgeWpsDueToGlobalReset			// Called after a global reset is done
// Overwrite in your stepping program implementation
END_METHOD

METHOD PROTECTED pauseAsNeeded : BOOL		// Will halt program execution when PAUSE is requested
oStopped := ic_isPauseByCsRequested() OR mIsPauseByManualRequested();
END_METHOD

METHOD PROTECTED pauseAsNeededByExternalRequest		// Pausing possibility from an external request
VAR_INPUT
	iExternalPauseRequest:	BOOL;
END_VAR
oStopped := iExternalPauseRequest;
END_METHOD

METHOD PROTECTED pauseAsNeededWithConditionCache : BOOL		// Will halt program execution when PAUSE is requested
															// Enables caching of iCondition in gotoNextStep
oStopped := ic_isPauseByCsRequested() OR mIsPauseByManualRequested();

enableConditionCache();
END_METHOD

METHOD PRIVATE setConditionCache : BOOL
VAR_INPUT
	iCondition:		BOOL;
	iReason:		T_SHORT_STR;
END_VAR
IF (iCondition AND conditionCacheActive AND NOT conditionCache) THEN
	conditionCache := TRUE;
	FC_GetLogger().info(iData := FC_4strConcat(iStr1:= getLoggingId(), iStr2 := ', ', iStr3 := iReason, iStr4 := oDebugStep));
END_IF
END_METHOD

METHOD PUBLIC stepAsString : T_SHORT_STR	// Return your ENUM step as STRING
forceMethodOverwrite(instancePath);
END_METHOD

METHOD PROTECTED stepInBetween : BOOL	// Returns TRUE if the current step is in between (=> and <=) Start and End step
VAR_INPUT
	iStart:	INT;	// Start step (inclusive)
	iEnd:	INT;	// End step (inclusive)
END_VAR
IF (stepPtr <> IING.ZERO_POINTER) THEN
	stepInBetween := (stepPtr^ >= iStart) AND (stepPtr^ <= iEnd);
ELSE
	stepInBetween := FALSE;
END_IF
END_METHOD

METHOD PRIVATE trace : BOOL
VAR_INPUT
	iLogTraces:		BOOL;
	iExtraTrace:	T_SHORT_STR;
END_VAR
VAR
	identifier:	T_SHORT_STR;
END_VAR
IF (stepChanged AND iLogTraces) THEN
	IF (FC_StringNotEmpty(iExtraTrace)) THEN
		identifier := FC_2strConcatSeparator(iSeparator := IING.STRING_UNDERSCORE, iStr1 := getLoggingId(), iStr2 := iExtraTrace);
	ELSE
		identifier := getLoggingId();
	END_IF

	// Do not use oDebugStep here since it gets updated only every xxx ms
	FC_GetLogger().trace(iData := FC_4strConcat(iStr1 := identifier, iStr2 := ', ', iStr3 := 'Step: ', iStr4 := stepAsString()));
END_IF
END_METHOD

METHOD PRIVATE updateOldStep : BOOL
IF (stepPtr^ <> oldStepForStepChangeOnly) THEN
	stepChanged := TRUE;
	prevStep := oldStepForStepChangeOnly;			// Otherwise next SWITCH CASE checks oldStep which was just updated here!!
	oldStepForStepChangeOnly := stepPtr^;
				
	stepStartedTime := TIME();
ELSE 
	stepChanged := FALSE;
END_IF
END_METHOD

END_FUNCTION_BLOCK

// ---- BASE/Misc/FB_BaseWithAlarmEvents.TcPOU
FUNCTION_BLOCK FB_BaseWithAlarmEvents EXTENDS FB_Base		// Base block providing alarm and forcing functions
VAR
//	alarmEvent:					FB_AlarmEvent;
//	warningEvent:				FB_WarningEvent;
	
//	forceEvent:					FB_ForceEvent;
END_VAR

METHOD PROTECTED forceMethodOverwrite : BOOL
VAR_INPUT
	iCaller: T_SHORT_STR;
END_VAR
FC_GetLogger().info(FC_2strConcatSeparator(iSeparator := IING.STRING_SPACE, iStr1 := 'Overwrite this method: ', iStr2 := iCaller));
END_METHOD

END_FUNCTION_BLOCK

// ---- BASE/Misc/FB_Base.TcPOU
FUNCTION_BLOCK FB_Base		// Base block providing Controls signals and Loggers
VAR_INPUT
	iControlSignals:			ST_CONTROL_SIGNALS_OUT;

	iPos:						E_POS := E_POS.UNDEFINED;
	iDeviceType:				E_DEVICE_TYPE := E_DEVICE_TYPE.CONVEYOR;
	iDeviceId:					T_DEVICE_ID := IING.STRING_BLANK;
	
	iControlSignalsIf:			I_ControlSignals;
END_VAR

METHOD PROTECTED forceMethodOverwrite : BOOL
VAR_INPUT
	iCaller: T_SHORT_STR;
END_VAR
FC_GetLogger().info(FC_2strConcatSeparator(iSeparator := IING.STRING_SPACE, iStr1 := 'Overwrite this method: ', iStr2 := iCaller));
END_METHOD

METHOD PUBLIC getLoggingId : T_SHORT_STR	// Returns DeviceType__Position.Id
getLoggingId := FC_GetLoggingId(iPos, iDeviceType, iDeviceId, IING.STRING_BLANK);
END_METHOD

METHOD PUBLIC getPositionWithId : T_SHORT_STR		// Returns Position.Id
getPositionWithId := FC_GetPositionWithId(iPos, iDeviceId);
END_METHOD

METHOD PUBLIC getPosNrWithId : T_SHORT_STR		// Returns Position.Id
getPosNrWithId := FC_GetPosNrWithId(iPos, iDeviceId);
END_METHOD

END_FUNCTION_BLOCK

// ---- LOGGING/FC_GetLogger.TcPOU
FUNCTION FC_GetLogger : I_Logger		// Gets the deault logger instance

// At PLC start and before cycleStart is called, the default Logger can be NULL, can cause a NULL pointer exception (eg. File logging instance before cycleStart and control signals calls logging) 
IF (LOGGER.defaultLogger <> 0) THEN
	FC_GetLogger := LOGGER.defaultLogger;
ELSE
	FC_GetLogger := LOGGER.nullLogger;
END_IF

END_FUNCTION

// ---- ALARMS/AppSupport/FC_GetLoggingId.TcPOU
FUNCTION FC_GetLoggingId : T_SHORT_STR		// Returns the ID of the given FB instance based on position, device type and extra field
VAR_INPUT
	iPos:			E_POS;
	iDeviceType:	E_DEVICE_TYPE;
	iDeviceId:		T_DEVICE_ID;
	iExtra:			T_SHORT_STR;
END_VAR

IF (FC_StringEmpty(iExtra)) THEN
	FC_GetLoggingId := FC_2strConcatSeparator(iSeparator := '__', iStr1 := TO_STRING(iDeviceType), iStr2 := FC_GetPositionWithId(iPos, iDeviceId));
ELSE
	FC_GetLoggingId := FC_3strConcatSeparator(iSeparator := '__', iStr1 := TO_STRING(iDeviceType), iStr2 := FC_GetPositionWithId(iPos, iDeviceId), iExtra);
END_IF

END_FUNCTION

// ---- BASE/StringUtils/FC_StringEmpty.TcPOU
FUNCTION FC_StringEmpty : BOOL	// Returns TRUE if the specified string length is more or equal to 1 
VAR_INPUT
	iString:	T_DEFAULT_STR;
END_VAR

FC_StringEmpty := LEN(iString) = 0;

END_FUNCTION

// ---- ALARMS/AppSupport/FC_GetPositionWithId.TcPOU
FUNCTION FC_GetPositionWithId : T_SHORT_STR
VAR_INPUT
	iPos:						E_POS := E_POS.UNDEFINED;
	iDeviceId:					T_DEVICE_ID := IING.STRING_BLANK;
END_VAR

FC_GetPositionWithId := FC_2strConcatSeparator(iSeparator := IING.STRING_DOT, iStr1 := TO_STRING(iPos), iStr2 := iDeviceId);

END_FUNCTION

// ---- ALARMS/AppSupport/FC_GetPosNrWithId.TcPOU
FUNCTION FC_GetPosNrWithId : T_SHORT_STR		// Returns the position number as INT followed by the ID
VAR_INPUT
	iPos:						E_POS := E_POS.UNDEFINED;
	iDeviceId:					T_DEVICE_ID := IING.STRING_BLANK;
END_VAR
VAR
	enumAsInt:					INT;	// INT_TO_STRING(ofAnEnum) prints the whole ENUM
END_VAR

enumAsInt := iPos;
FC_GetPosNrWithId := FC_2strConcatSeparator(iSeparator := IING.STRING_DOT, iStr1 := INT_TO_STRING(enumAsInt), iStr2 := iDeviceId);

END_FUNCTION

// ---- BASE/Misc/FB_BoolLogger.TcPOU
FUNCTION_BLOCK FB_BoolLogger EXTENDS FB_BoolTrigger		// Logs the changes in a BOOL signal, usefull for logging a DI
VAR_INPUT
	iLogRising:		BOOL := FALSE;
	iLogFalling:	BOOL := FALSE;
	iLogLevel:		E_LOG_LEVEL := E_LOG_LEVEL.TRACE;
END_VAR

SUPER^(iIn := iIn);

IF (iLogRising AND oRTrig) THEN
	FC_GetLogger().doLog(iData := FC_2strConcatSeparator(iSeparator := IING.STRING_BLANK, iStr1 := 'Rising edge:', iStr2 := getLoggingId()), iLogLevel);
END_IF

IF (iLogFalling AND oFTrig) THEN
	FC_GetLogger().doLog(iData := FC_2strConcatSeparator(iSeparator := IING.STRING_BLANK, iStr1 := 'Falling edge:', iStr2 := getLoggingId()), iLogLevel);
END_IF

END_FUNCTION_BLOCK

// ---- BASE/Misc/FB_BoolTrigger.TcPOU
FUNCTION_BLOCK FB_BoolTrigger EXTENDS FB_Base		// Detects rising and falling edges on the input
VAR_INPUT
	iIn:			BOOL;
END_VAR
VAR_OUTPUT
	oRtrig:			BOOL;
	oFtrig:			BOOL;
	oChanged:		BOOL;
END_VAR
VAR
	rTrig:			R_TRIG;
	fTrig:			F_TRIG;
END_VAR

rTrig(CLK := iIn, Q => oRtrig);
fTrig(CLK := iIn, Q => oFtrig);

oChanged := oRtrig OR oFtrig;

END_FUNCTION_BLOCK

// ---- BASE/StringUtils/FC_4strConcat.TcPOU
FUNCTION FC_4strConcat : T_DEFAULT_STR		// Concatenates 4 strings
VAR_INPUT
	iStr1:		T_DEFAULT_STR;
	iStr2:		T_DEFAULT_STR;
	iStr3:		T_DEFAULT_STR;
	iStr4:		T_DEFAULT_STR;
END_VAR

FC_4strConcat := CONCAT(FC_3strConcat(iStr1, iStr2, iStr3), iStr4);

END_FUNCTION

// ---- BASE/ControlSignals/FB_ControlSignalResets.TcPOU
FUNCTION_BLOCK FB_ControlSignalResets
VAR_INPUT
	iReset:						BOOL;	// Manually pressed the reset button
	iExternalReset:				BOOL;	// Reset came through FB input, eg. hard wired button/banner reset
	iHardreset:					BOOL;	
	iAutoReset:					BOOL;	// Reset came through FB input due to some automated process (eg. SA doors closed)
	
	iPos:						E_POS;
	iMiscArea:						T_SHORT_STR;	// Misc area in case iPos does not fit well.  Must be from TM_Devices.E_SAFETY_AREA or TM_Base.E_MISC_AREAS. 
END_VAR
VAR_OUTPUT
	oResetPulse:				BOOL;
	oHardResetPulse: 			BOOL;
	
	oExtendedResetPulse:		BOOL;	// Extended reset pulse for external systems
	oExtendedHardResetPulse:	BOOL;	// Extended reset pulse for external systems
END_VAR
VAR_IN_OUT
	ioStaticSettings:					ST_CONTROL_SIGNALS_STATIC_SETTINGS;
END_VAR
VAR
	resetDelay:						TON;
	externalResetDelay:				TON;
	hardResetDelay:					TON;

	resetPulse:						R_TRIG;
	autoResetPulse:					R_TRIG;
	externalResetPulse:				R_TRIG;

	hardResetPulse:					R_TRIG;
	extendedResetPulseDelay:		TOF;
	extendedHardResetPulseDelay:	TOF;
END_VAR

resetDelay(IN := iReset, PT := ioStaticSettings.resetTime);
externalResetDelay(IN := iExternalReset, PT := ioStaticSettings.resetTime);
hardResetDelay(IN := iHardReset, PT := ioStaticSettings.hardResetTime);

resetPulse(CLK := resetDelay.Q);
autoResetPulse(CLK := iAutoReset);
externalResetPulse(CLK := externalResetDelay.Q);


oResetPulse := resetPulse.Q OR autoResetPulse.Q OR externalResetPulse.Q;

hardResetPulse(CLK := hardResetDelay.Q, Q => oHardResetPulse);

extendedResetPulseDelay(IN := oResetPulse, PT := ioStaticSettings.extendedResetPulseDuration, Q => oExtendedResetPulse);
extendedHardResetPulseDelay(IN := oHardResetPulse, PT := ioStaticSettings.extendedResetPulseDuration, Q => oExtendedHardResetPulse);

IF (resetPulse.Q) THEN
	FC_GetDataReporter().ic_resetDone(iPos, iMiscArea, E_RESET_ORIGIN.CONTROL_AREA_MANUAL, IING.STRING_BLANK);
END_IF;

IF (autoResetPulse.Q) THEN
	FC_GetDataReporter().ic_resetDone(iPos, iMiscArea, E_RESET_ORIGIN.CONTROL_AREA_AUTO, IING.STRING_BLANK);
END_IF

IF (externalResetPulse.Q) THEN
	FC_GetDataReporter().ic_resetDone(iPos, iMiscArea, E_RESET_ORIGIN.EXTERNAL, IING.STRING_BLANK);
END_IF;

END_FUNCTION_BLOCK

// ---- DATA/REPORTING/FC_GetDataReporter.TcPOU
FUNCTION FC_GetDataReporter : I_DataReporter		// Helper function returning an instance of 'a' data reporter
	// If no real implementation is available, a dummy/stub implementation will be returned

IF (DATA_REPORTER_BASE.defaultReporter <> 0) THEN
	FC_GetDataReporter := DATA_REPORTER_BASE.defaultReporter;
ELSE
	FC_GetDataReporter := DATA_REPORTER_BASE.dummyReporter;
END_IF

END_FUNCTION

// ---- BASE/ControlSignals/FB_ControlSignalsV2.TcPOU
FUNCTION_BLOCK FB_ControlSignalsV2 IMPLEMENTS I_ControlSignals	// Handles the control signal inputs (auto/manual/service/reset/hard reset) for use in our application
VAR_INPUT
	iExternalReset:					BOOL := FALSE;				// External reset, eg. banner reset
	iExternalPauseRequest:			BOOL := FALSE;				// Pause request, eg. from doors/button box
	
//	iExternalControlSignals:		POINTER TO ST_CONTROL_SIGNALS_V2;	// Used by conveyors (having internal control signals)
	
	iAutoReset:						BOOL := FALSE;				// Intended to be used in AUTO mode, no delays in here
	iSaOkDelayed:					BOOL;						// Used to pause/unpause
	
	iExternalAutoPtr:				POINTER TO BOOL;			// Hardwired Auto switch (Packing BB400)
	iIgnoreCycleStart:				BOOL := FALSE;				// When ignored, state wont go to manual at startup
	iPos:							E_POS := E_POS.UNDEFINED;
	iMiscArea:						T_SHORT_STR;	// Misc area in case iPos does not fit well.  Must be from TM_Devices.E_SAFETY_AREA or TM_Base.E_MISC_AREAS. 
END_VAR
VAR_OUTPUT
	{ attribute 'TcHmiSymbol.Show' }
	oControlSignals:				POINTER TO ST_CONTROL_SIGNALS_V2;
END_VAR
VAR_IN_OUT
	ioTcHmi:	TC_HMI_CS;
END_VAR
VAR
	{ attribute 'TcHmiSymbol.ShowRecursively' }
	controlSignals:					ST_CONTROL_SIGNALS_V2;
	previousCs:						ST_CONTROL_SIGNALS_OUT;
	reset:							BOOL;
	externalReset:					BOOL;
	autoReset:						BOOL;
	hardReset:						BOOL;
	stopImmediately:				BOOL;
	resets:							FB_ControlSignalResets;
	stopImmediatelyPulse:			R_TRIG;
	
	autoBoolTrigger:				FB_BoolTrigger;
	manualBoolTrigger:				FB_BoolTrigger;
	serviceBoolTrigger:				FB_BoolTrigger;
	pauseRequestBoolTrigger:		FB_BoolTrigger;
	
	serviceTimer:					TON;
	externalPauseRequestTrigger:	FB_BoolTrigger;
	saOkTrigger:					FB_BoolTrigger;
	
	
	manualButtonTriggers:			FB_BoolTrigger;
	
	externalAuto:					BOOL;
	externalManual:					BOOL;
	externalAutoTrigger:			FB_BoolTrigger;
	failingToSwitchToAuto:			BOOL;
	
//	warningEvent:					FB_WarningEvent;
//	alarmEvent:						FB_AlarmEvent;
END_VAR
VAR PERSISTENT
	{ attribute 'TcHmiSymbol.Show' }
	settings:						ST_CONTROL_SIGNALS_SETTINGS;
END_VAR
VAR_STAT PERSISTENT
	{ attribute 'TcHmiSymbol.Show' }
	staticSettings:					ST_CONTROL_SIGNALS_STATIC_SETTINGS;
END_VAR

// ---------------------------------------------- HMI
controlSignals.in := ioTcHmi.in;


controlsignals.settings REF= settings;
controlsignals.staticSettings REF= staticSettings;

externalPauseRequestTrigger(iIn := iExternalPauseRequest);
saOkTrigger(iIn := iSaOkDelayed);

// When BBs request to enter, iExternalPauseRequest goes ON and we set the PAUSE signal here ONCE
// When the safety area goes down, we pause
// Triggers are used here so that the HMI buttons keep working
IF (externalPauseRequestTrigger.oRtrig OR saOkTrigger.oFtrig) THEN
	controlSignals.in.pauseRequest := TRUE;
END_IF

// If doors are closed and safety is OK, pause is switched OFF (eg. pressing BB pause request and then cancelling it)
// When the safety area goes ok, we take away the pause request
IF ((externalPauseRequestTrigger.oFtrig AND iSaOkDelayed) OR saOkTrigger.oRtrig) THEN
	controlSignals.in.pauseRequest := FALSE;
END_IF


	manualButtonTriggers(iIn := controlSignals.in.manualMode);


	// Service mode is switched back OFF
	IF (serviceTimer.Q) THEN
		controlSignals.in.serviceMode := FALSE;
	END_IF	

	// Toggle
	IF (manualButtonTriggers.oRtrig) THEN
		controlSignals.out.manual := NOT controlSignals.out.manual;
	END_IF
	
	IF (NOT iIgnoreCycleStart AND IING.cycleStart) THEN
		controlSignals.out.manual := TRUE;
	END_IF
	
	controlSignals.out.auto := NOT controlSignals.out.manual;

	controlSignals.out.service := controlSignals.in.serviceMode;
	controlSignals.out.pauseRequest := controlSignals.in.pauseRequest;

	reset := controlSignals.in.reset;
	externalReset := controlSignals.in.externalReset;
	
	autoReset := controlSignals.in.autoReset;
	hardreset := controlSignals.in.hardReset;
	stopImmediately := controlSignals.in.stopImmediately;


autoBoolTrigger(iIn := controlSignals.out.auto, oRtrig => controlSignals.out.autoPulse, oFtrig => controlSignals.out.autoOffPulse);
manualBoolTrigger(iIn := controlSignals.out.manual, oRtrig => controlSignals.out.manualPulse, oFtrig => controlSignals.out.manualOffPulse);
serviceBoolTrigger(iIn := controlSignals.out.service, oRtrig => controlSignals.out.servicePulse, oFtrig => controlSignals.out.serviceOffPulse);
pauseRequestBoolTrigger(iIn := controlSignals.in.pauseRequest);

// Switching OFF service mode automatically after a delay
serviceTimer(IN := controlSignals.out.service, PT := staticSettings.serviceResetTime);

stopImmediatelyPulse(CLK := stopImmediately, Q => controlSignals.out.stopImmediately); 

// Hard reset is only possible in service mode
resets(iReset := reset,	iExternalReset := externalReset,
	iHardreset := controlSignals.out.manual AND controlSignals.out.service AND hardReset,
	iAutoReset := autoReset, iPos := iPos, iMiscArea := iMiscArea, ioStaticSettings := staticSettings,
	oResetPulse => controlSignals.out.resetPulse, oHardResetPulse => controlSignals.out.hardResetPulse,
	oExtendedResetPulse => controlSignals.out.extendedResetPulse,
	oExtendedHardResetPulse => controlSignals.out.extendedHardResetPulse);

oControlSignals := ADR(controlSignals);

// External signals are set into this structure which makes it possible to pass as 'iExternalControlSignals'
controlSignals.in.externalReset := iExternalReset;
controlSignals.in.autoReset := iAutoReset;

mCheckValues();
aReportingAndLogging();
//mInitializeName(IIN.pulse10S);

// Old value for data collection purposes
previousCs := controlSignals.out;

aExternalSwitch();
aHmi();
mWarningsAndAlarms();


ioTcHmi.out := controlSignals.out;

ACTION aExternalSwitch:
IF (iExternalAutoPtr <>  IING.ZERO_POINTER) THEN
	// Dereference the pointer
	externalAuto := iExternalAutoPtr^;
	externalManual := NOT externalAuto;
	
	// Trying to switch to Auto but external is still in Manual
	failingToSwitchToAuto := externalManual AND controlSignals.in.manualMode;

	// Rising/falling edge detection
	externalAutoTrigger(iIn := externalAuto);

	// External manual always forces the control signal to Manual
	IF (externalManual) THEN
		controlSignals.out.manual := TRUE;
	END_IF
	
	// External switched to Auto
	IF (externalAutoTrigger.oRtrig) THEN
		controlSignals.out.manual := FALSE;
	END_IF

ELSE
	externalAuto := TRUE;
	externalManual := NOT externalAuto;
END_IF
END_ACTION

ACTION aHmi:
controlSignals.out.externalManualActive := externalManual;
controlSignals.out.failingToSwitchToAuto := failingToSwitchToAuto;
END_ACTION

ACTION aReportingAndLogging:
IF (controlSignals.out.autoPulse) THEN
	FC_GetLogger().debug(FC_3strConcatSeparator(iSeparator := IING.STRING_SPACE, iStr1 := TO_STRING(iPos), iStr2 := settings.name, iStr3 := ' switched to AUTO'));
	FC_GetDataReporter().ic_operationModeChanged(iPos, iMiscArea, E_OPERATION_MODE.AUTO);
END_IF
IF (controlSignals.out.manualPulse) THEN
	FC_GetLogger().debug(FC_3strConcatSeparator(iSeparator := IING.STRING_SPACE, iStr1 := TO_STRING(iPos), iStr2 := settings.name, iStr3 := ' switched to MANUAL'));
	FC_GetDataReporter().ic_operationModeChanged(iPos, iMiscArea, E_OPERATION_MODE.MANUAL);
END_IF

IF (controlSignals.out.servicePulse) THEN
	FC_GetLogger().debug(FC_3strConcatSeparator(iSeparator := IING.STRING_SPACE, iStr1 := TO_STRING(iPos), iStr2 := settings.name, iStr3 := ' switched to SERVICE'));
	FC_GetDataReporter().ic_serviceStateChanged(iPos, iMiscArea, TRUE);
END_IF
IF (controlSignals.out.serviceOffPulse) THEN
	FC_GetLogger().debug(FC_3strConcatSeparator(iSeparator := IING.STRING_SPACE, iStr1 := TO_STRING(iPos), iStr2 := settings.name, iStr3 := ' switched to SERVICE OFF'));
	FC_GetDataReporter().ic_serviceStateChanged(iPos, iMiscArea, FALSE);
END_IF

IF (controlSignals.out.resetPulse) THEN
	FC_GetLogger().info(FC_3strConcatSeparator(iSeparator := IING.STRING_SPACE, iStr1 := TO_STRING(iPos), iStr2 := settings.name, iStr3 := ' reset pulse'));
	
	// Data reporting in FB_ControlSignalResets and FB_EventResetHandler and
END_IF

IF (controlSignals.out.hardResetPulse) THEN
	FC_GetLogger().info(FC_3strConcatSeparator(iSeparator := IING.STRING_SPACE, iStr1 := TO_STRING(iPos), iStr2 := settings.name, iStr3 := ' hard reset pulse'));
	FC_GetDataReporter().ic_initializeDone(iPos, iMiscArea, E_RESET_ORIGIN.CONTROL_AREA_MANUAL);
END_IF

IF (pauseRequestBoolTrigger.oRtrig) THEN
	FC_GetLogger().debug(FC_3strConcatSeparator(iSeparator := IING.STRING_SPACE, iStr1 := TO_STRING(iPos), iStr2 := settings.name, iStr3 := ' pause requested'));
END_IF

IF (pauseRequestBoolTrigger.oFtrig) THEN
	FC_GetLogger().debug(FC_3strConcatSeparator(iSeparator := IING.STRING_SPACE, iStr1 := TO_STRING(iPos), iStr2 := settings.name, iStr3 := ' pause request OFF'));
END_IF
END_ACTION

METHOD ic_getControlSignalsOutPtr : POINTER TO ST_CONTROL_SIGNALS_OUT
ic_getControlSignalsOutPtr := ADR(controlSignals.out);
END_METHOD

METHOD PUBLIC ic_getControlSignalsPtr : POINTER TO ST_CONTROL_SIGNALS_V2
ic_getControlSignalsPtr := oControlSignals;
END_METHOD

METHOD PUBLIC ic_isInAuto : BOOL
ic_isInAuto := controlSignals.out.auto;
END_METHOD

METHOD public ic_isInPause : BOOL
ic_isInPause := controlSignals.out.pauseRequest;
END_METHOD

METHOD PUBLIC ic_switchToAuto
FC_GetLogger().debug(FC_3strConcatSeparator(iSeparator := IING.STRING_SPACE, iStr1 := TO_STRING(iPos), iStr2 := settings.name, iStr3 := ' asked to switched to AUTO'));


	controlSignals.out.manual := FALSE;
END_METHOD

METHOD PUBLIC ic_unPause
FC_GetLogger().debug(FC_3strConcatSeparator(iSeparator := IING.STRING_SPACE, iStr1 := TO_STRING(iPos), iStr2 := settings.name, iStr3 := ' asked to UN-pause'));

	controlSignals.in.pauseRequest := FALSE;
END_METHOD

METHOD PRIVATE mCheckValues : BOOL
// It can happen that the hard reset time becomes smaller (or 0) than the reset time, either by accident
// or when memory shift during download messes up

// When this happens it may be impossible to open up the service menu (since the service timer expires too fast)
//  To prevent problems, the defaults get restored when this happens

IF ((staticSettings.hardResetTime < staticSettings.resetTime) OR (staticSettings.resetTime = T#0S)) THEN
	staticSettings.resetTime := IING.RESET_TIME;
	staticSettings.hardResetTime := IING.HARD_RESET_TIME;
	staticSettings.serviceResetTime := IING.AUTO_SERVICE_RESET_TIME;
	staticSettings.extendedResetPulseDuration := IING.EXTENDED_RESET_PULSE_DURATION;
END_IF
END_METHOD

METHOD PRIVATE mInitializeName : BOOL
VAR_INPUT
	iCondition:		BOOL;
END_VAR
VAR
	enumAsInt:					INT;	// INT_TO_STRING(ofAnEnum) prints the whole ENUM
END_VAR
IF (iCondition) THEN
	enumAsInt := iPos;
	settings.name := INT_TO_STRING(enumAsInt);
END_IF
END_METHOD

METHOD mWarningsAndAlarms	// Create warning when external manual is forced
							// Create alarm when external manual is forced and trying to switch to Automatic
END_METHOD

END_FUNCTION_BLOCK

// ---- BASE/CycleStartEnd/FB_CycleEnd.TcPOU
FUNCTION_BLOCK FB_CycleEnd		// Must always be the last call in PLC MAIN, does necessary things needed in every project
VAR
END_VAR

END_FUNCTION_BLOCK

// ---- BASE/CycleStartEnd/FC_GetCurrentCycleCount.TcPOU
FUNCTION FC_GetCurrentCycleCount : UDINT

FC_GetCurrentCycleCount := IING.cycleCounter;

END_FUNCTION

// ---- BASE/FileUtils/FC_FilePathGenerator.TcPOU
FUNCTION FC_FilePathGenerator : T_MaxString
VAR_INPUT
	iPath:			T_MaxString;
	iFile:			T_MaxString;
END_VAR

FC_FilePathGenerator := FC_3strConcat(iStr1 := iPath, iStr2 := IING.STRING_BACKSLASH, iStr3 := iFile);

END_FUNCTION

// ---- BASE/LocaleUtils/FB_TimeSync.TcPOU
FUNCTION_BLOCK FB_TimeSync		// FB for synchronizing the PLC times from the 'master/main', a maximum of 10 slaves can be synchronized
VAR_INPUT	
	iAmsNetIds:				POINTER TO T_AmsNetID;		// Ams net id of the slaves we want to time sync
	iAmsNetIdArraySize:		INT;						// Number of Ams net ids passed (= the array size)
	iSyncInterval: 			TIME;						// Time interval between synchronizations
END_VAR
VAR
	pulser:					FB_Pulse;										// Pulser for starting the time sync
	fbNtSetLocalTime:		ARRAY[0..MAX_SYNC_SIZE-1] OF NT_SetLocalTime;	// Memory reservation for max x slave syncing
	i: 						INT;											// For loop
	minCnt:					INT;
END_VAR
VAR CONSTANT
	MAX_SYNC_SIZE:			INT := 10;	// We can set a maximum of 10 slave PLCs here
END_VAR

pulser(iTime := iSyncInterval);

// We must prevent out of array bounds
minCnt := MIN(iAmsNetIdArraySize, MAX_SYNC_SIZE);
IF (minCnt > MAX_SYNC_SIZE) THEN
	minCnt := MAX_SYNC_SIZE;
END_IF

FOR i := 0 TO minCnt - 1 BY 1 DO
	fbNtSetLocalTime[i](NETID := iAmsNetIds[i], TIMESTR := IING.localSystemTime, START:= pulser.oPulse);	// IIN.localSystemTime is part of TM_Base
END_FOR

END_FUNCTION_BLOCK

// ---- BASE/LocaleUtils/FC_DateAndTimeToDt.TcPOU
FUNCTION FC_DateAndTimeToDt : DT		// Converts a Date/time string to 'DT', this is usefull for doing calculations on time
VAR_INPUT
	iDateAndTime:			T_SHORT_STR;	// Date and time as string
END_VAR
VAR
	timeStamp:				T_SHORT_STR;
	systemTime:				TIMESTRUCT;
	dateTime:				DT;
END_VAR

timeStamp := iDateAndTime;

timeStamp := FC_CharReplace(iString := timeStamp, iOrigChar := ',', iReplaceChar := '.');
timeStamp := FC_CharReplace(iString := timeStamp, iOrigChar := ' ', iReplaceChar := '-');

systemTime := STRING_TO_SYSTEMTIME(timeStamp);
FC_DateAndTimeToDt := SYSTEMTIME_TO_DT(systemTime);

END_FUNCTION

// ---- BASE/StringUtils/FC_CharReplace.TcPOU
FUNCTION FC_CharReplace : T_DEFAULT_STR		// Replaces a character inside a string with another character
VAR_INPUT
	iString:			T_DEFAULT_STR;		// String where a character is to be replaced
	iOrigChar:			T_SHORT_STR;		// Character to be replaced
	iReplaceChar:		T_SHORT_STR;		// Character we are replacing with
END_VAR
VAR
	charPos:			INT;
END_VAR

FC_CharReplace := iString;
charPos := find(STR1 := FC_CharReplace, STR2 := iOrigChar);
IF (charPos > 0) THEN
	FC_CharReplace := REPLACE(STR1 := FC_CharReplace, STR2 := iReplaceChar, L := 1, P := charPos);
END_IF

END_FUNCTION

// ---- BASE/LocaleUtils/FC_GetLocalDateAndTimeString.TcPOU
FUNCTION FC_GetLocalDateAndTimeString : T_SHORT_STR		// Returns the local date and time as string,  eg. '27:05:2019 15:58:40:302'. Use E_REGIO_SELECTION at FB_CycleStart for a different format.

FC_GetLocalDateAndTimeString := IING.localDateAndTimeString;

END_FUNCTION

// ---- BASE/LocaleUtils/FC_GetLocalDateString.TcPOU
FUNCTION FC_GetLocalDateString : T_SHORT_STR;		// Returns the local date string, eg. '27:5:2019'. Use E_REGIO_SELECTION at FB_CycleStart for a different format.

FC_GetLocalDateString := IING.localDateString;

END_FUNCTION

// ---- BASE/LocaleUtils/FC_GetLocalTimeString.TcPOU
FUNCTION FC_GetLocalTimeString : T_SHORT_STR		// Returns the local time as string, eg. '15:58:40:302'

FC_GetLocalTimeString := IING.localTimeString;

END_FUNCTION

// ---- BASE/LocaleUtils/FC_GetLocalTimeStringMinAccuracy.TcPOU
FUNCTION FC_GetLocalTimeStringMinAccuracy : T_SHORT_STR	// Returns the local time as short string, eg. '08:02 AM'.
													// Use E_REGIO_SELECTION at FB_CycleStart for a different format.

FC_GetLocalTimeStringMinAccuracy := IING.localTimeMinAccuracy;

END_FUNCTION

// ---- BASE/LocaleUtils/FC_GetLocalTimeStringSecAccuracy.TcPOU
FUNCTION FC_GetLocalTimeStringSecAccuracy : T_SHORT_STR	// Returns the local time as short string, eg. '08:02:21 AM'.
													// Use E_REGIO_SELECTION at FB_CycleStart for a different format.

FC_GetLocalTimeStringSecAccuracy := IING.localTimeSecAccuracy;

END_FUNCTION

// ---- BASE/LocaleUtils/FC_GetUsDateString.TcPOU
FUNCTION FC_GetUsDateString : T_SHORT_STR;		// Returns the US date string, especially usefull for naming log files

FC_GetUsDateString := IING.usDateString;

END_FUNCTION

// ---- BASE/LocaleUtils/FC_NowAsDt.TcPOU
FUNCTION FC_NowAsDt : DT		// Returns the current time (=now) as 'DT'

FC_NowAsDt := FC_DateAndTimeToDt(iDateAndTime := FC_GetLocalDateAndTimeString());

END_FUNCTION

// ---- BASE/LocaleUtils/FC_TimeStringToDt.TcPOU
FUNCTION FC_TimeStringToDt : DT		// Converts a time string to 'DT', this is usefull for doing calculations on time
VAR_INPUT
	iTime:				T_SHORT_STR;		// Time as string
END_VAR
VAR
	timeStamp:			T_SHORT_STR;
END_VAR

timeStamp := FC_GetLocalDateString();
timeStamp := FC_2strConcatSeparator(iSeparator := ' ', iStr1 := timeStamp, iStr2 := iTime);

FC_TimeStringToDt := FC_DateAndTimeToDt(iDateAndTime := timeStamp);

END_FUNCTION

// ---- BASE/Misc/FB_DelayedReset.TcPOU
FUNCTION_BLOCK FB_DelayedReset		// Delays (hard) reset pulse
									// Robot main sequence should wait doing hard reset until sub sequences have gotten it 
VAR_INPUT
	iReset:						BOOL;
	iDelay:						TIME := T#100MS;	// After this delay, reset pulse (1 PLC cycle) will be given
END_VAR
VAR_OUTPUT
	oDelayedResetPulse:			BOOL;
END_VAR
VAR
	resetCame:					BOOL;
	resetDelay:					TON;
	resetDelayEdge:				R_TRIG;
END_VAR

IF (iReset) THEN
	resetCame := TRUE;
END_IF

resetDelay(IN := resetCame, PT := iDelay);
resetDelayEdge(CLK := resetDelay.Q);

IF (resetDelayEdge.Q) THEN
	resetCame := FALSE;
END_IF

oDelayedResetPulse := resetDelayEdge.Q;

END_FUNCTION_BLOCK

// ---- BASE/Misc/FB_HandshakeDelay.TcPOU
FUNCTION_BLOCK FB_HandshakeDelay	// Delays the signal (TOF) so the handshake has enough time to be seen by the other part (inside PLC/EAP/normal IO)
VAR_INPUT
	iHandshake:			BOOL;				// The handshake signal
	iSignalDuration:	TIME := T#100MS;	// The delay
END_VAR
VAR_OUTPUT
	oHandshake:	BOOL;						// The handshake signal having an additional delay
END_VAR
VAR
	delay: TOF;
END_VAR

delay(IN := iHandshake, PT := iSignalDuration, Q => oHandshake);

END_FUNCTION_BLOCK

// ---- BASE/Misc/FB_IntChangeTrigger.TcPOU
FUNCTION_BLOCK FB_IntChangeTrigger EXTENDS FB_Base	// Monitors an INTEGER and sets a 1 PLC cycle flag when changed
VAR_INPUT
	iInt:			INT;
END_VAR
VAR_OUTPUT
	oChanged:		BOOL;	// TRUE (1 PLC cycle) when iInt has changed
	oOld:			INT;	// The value before the change
	oNew:			INT;	// The new (up to date) value
END_VAR
VAR
	old:			INT;
END_VAR

oNew := iInt;
oChanged := (old <> oNew);
old := iInt;

IF (NOT oChanged) THEN
	oOld := old;
END_IF

END_FUNCTION_BLOCK

// ---- BASE/Misc/FB_IntLogger.TcPOU
FUNCTION_BLOCK FB_IntLogger EXTENDS FB_IntChangeTrigger		// Logs the changes in an INT signal
VAR_INPUT
	iLogLevel:		E_LOG_LEVEL := E_LOG_LEVEL.TRACE;
END_VAR

SUPER^(iInt := iInt);

IF (oChanged) THEN
	FC_GetLogger().doLog(iData := FC_5strConcatSeparator(iSeparator := IING.STRING_BLANK, iStr1 := getLoggingId(), iStr2 := ' changed from old: ',
		iStr3 := INT_TO_STRING(oOld), iStr4 := ', New: ', iStr5 := INT_TO_STRING(oNew)), iLogLevel);
END_IF

END_FUNCTION_BLOCK

// ---- BASE/StringUtils/FC_5strConcatSeparator.TcPOU
FUNCTION FC_5strConcatSeparator : T_DEFAULT_STR		// Concatenates 5 strings with given separator
VAR_INPUT
	iSeparator:		STRING := IING.STRING_UNDERSCORE;
	iStr1:			T_DEFAULT_STR;
	iStr2:			T_DEFAULT_STR;
	iStr3:			T_DEFAULT_STR;
	iStr4:			T_DEFAULT_STR;
	iStr5:			T_DEFAULT_STR;
END_VAR

FC_5strConcatSeparator := FC_2strConcatSeparator(iSeparator := iSeparator,
	iStr1 := FC_4strConcatSeparator(iSeparator := iSeparator, iStr1 := iStr1, iStr2 := iStr2, iStr3 := iStr3, iStr4 := iStr4), iStr2 := iStr5);

END_FUNCTION

// ---- BASE/StringUtils/FC_4strConcatSeparator.TcPOU
FUNCTION FC_4strConcatSeparator : T_DEFAULT_STR		// Concatenates 4 strings with given separator
VAR_INPUT
	iSeparator:		STRING := IING.STRING_UNDERSCORE;
	iStr1:			T_DEFAULT_STR;
	iStr2:			T_DEFAULT_STR;
	iStr3:			T_DEFAULT_STR;
	iStr4:			T_DEFAULT_STR;
END_VAR

FC_4strConcatSeparator := FC_2strConcatSeparator(iSeparator := iSeparator,
	iStr1 := FC_3strConcatSeparator(iSeparator := iSeparator, iStr1 := iStr1, iStr2 := iStr2, iStr3 := iStr3), iStr2 := iStr4);

END_FUNCTION

// ---- BASE/Misc/FB_MemoryMonitor.TcPOU
FUNCTION_BLOCK FB_MemoryMonitor		// Will read the Router info periodically and log the available memory
VAR_INPUT
	iPulser:		BOOL;			// Put a periodic PULSER (1 plc cycle high) here
END_VAR
VAR
	getRouterStatusInfo:		FB_GetRouterStatusInfo;
	statusInfoReadyEdge:		R_TRIG;
	statusInfo:					ST_TcRouterStatusInfo;
	totalMem:					DINT;
	freeMem:					DINT;
END_VAR

getRouterStatusInfo(bExecute := iPulser, tTimeout := IING.ADS_WRITE_TIMEOUT, info => statusInfo);

